			IF fbListClosed.LUIDInList(ipEachPathAhead.StationDestination.LUID) THEN
				// if the successor node is already on the closed list - do nothing, repeate WHILE loop
				CONTINUE;
			END_IF
			
			//Calculate distance to start oh the new found station
			fPathLength := ipActiveStationAStar.PathLength + ipEachPathAhead.Length;
		
			//Check if this station is allready existin in open list - compare if this one is shorter
			IF __QUERYINTERFACE( fbListOpen.FindLUID(ipEachPathAhead.StationDestination.LUID), ipPathFoundInOpenList)  THEN
				IF ipPathFoundInOpenList.PathLength <= fPathLength  THEN
					//object in open list is shorter - do nothing, repeate WHILE loop
					CONTINUE;
				ELSE
					//new object is shorter - remove old object in open lsit
					fbListOpen.RemoveObject(ipPathFoundInOpenList);
				END_IF
			END_IF			
			
			
			//Add this path ahead to open list - set new length
			__QUERYINTERFACE(fbListNotUsedNodes.GetNextObject(), ipEmptyPathObj);
			ipEmptyPathObj.Station := ipEachPathAhead.StationDestination;
			ipEmptyPathObj.RouteUsedToNode.Duplicate(ipActiveStationAStar.RouteUsedToNode);
			ipEmptyPathObj.RouteUsedToNode.AddObject(ipEachPathAhead);
			fbListOpen.AddObject(ipEmptyPathObj);

		END_WHILE
		ipActiveStationAStar.Station.PathsAhead.RestoreIterator();

	END_IF

END_WHILE


//Return station or nothing
IF ipBesStationAStar = 0 THEN
	GetPathToTarget := 0;
ELSE
	//store list in an instance
	fbLastFoundResult.Station := ipBesStationAStar.Station;
	fbLastFoundResult.RouteUsedToNode.Duplicate(ipBesStationAStar.RouteUsedToNode);
	GetPathToTarget := fbLastFoundResult;
END_IF
END_METHOD

METHOD PROTECTED GetPosOnTrack : HRESULT
VAR
	fbPositionXYC : PositionXYC;
END_VAR
//GetArcLengthClosestTo track
THIS^.fPositionOnTrack := THIS^.ipAccocietedTrack.PlanarTrack.GetArcLengthClosestTo(geometry:= THIS^.fbPositionPlanned);

//Get the XYC Pos on track
THIS^.ipAccocietedTrack.PlanarTrack.GetPositionAt(THIS^.PositionOnTrack, fbPositionXYC);

//XYC -> XY
THIS^.fbPositionOnTrackXY.SetValuesXY(fbPositionXYC.x,fbPositionXYC.y);


//Check for NaN
IF NOT(THIS^.fPositionOnTrack = THIS^.fPositionOnTrack) THEN
	GetPosOnTrack := E_FAIL;
	RETURN;
END_IF
END_METHOD

METHOD PROTECTED GetStationAhead : HRESULT
VAR
	ipPath 		: I_XP_Path;
END_VAR
fbStationsAhead.Clear();


fbListPathAhead.ResetIterator();
WHILE fbListPathAhead.HasNextObject() DO
	IF __QUERYINTERFACE(fbListPathAhead.GetNextObject(),ipPath) THEN
		//add StationDestination to list
		fbStationsAhead.AddObject(ipPath.StationDestination);
	END_IF
END_WHILE
END_METHOD

METHOD PROTECTED GetStationBehinde : HRESULT
VAR_INPUT
END_VAR
VAR
	ipThisStation : I_XP_Station;
	ipXpStation : I_XP_Station;
	ipXpStationAhead : I_XP_Station;
END_VAR
ipThisStation := THIS^;
fbStationsBehinde.Clear();

//Check each Station
THIS^.ipXpSystem.StationsUsed.ResetIterator();
WHILE THIS^.ipXpSystem.StationsUsed.HasNextObject() DO
	IF __QUERYINTERFACE(THIS^.ipXpSystem.StationsUsed.GetNextObject(),ipXpStation) THEN
		//check the list of stations ahead if this station one is existing
		ipXpStation.StationsAhead.ResetIterator();
		WHILE ipXpStation.StationsAhead.HasNextObject() DO
			IF __QUERYINTERFACE(ipXpStation.StationsAhead.GetNextObject(),ipXpStationAhead) AND_THEN (ipXpStationAhead = ipThisStation) THEN
				//add station to list
				fbStationsBehinde.AddObject(ipXpStation);
			END_IF
		END_WHILE	
	END_IF
END_WHILE	
THIS^.ipXpSystem.StationsUsed.RestoreIterator();
END_METHOD

METHOD Initialize : HRESULT
VAR
	ipEachStationAhead : I_XP_Station;
	nIdx : UDINT;
END_VAR
VAR_INST
	//This error cannot be reset. Requires a reset cold
	{attribute 'hide'}	
	fbInitError : FB_TcAlarm;
	{attribute 'hide'}	
	fbMissingInterfaceAlarm : FB_TcAlarm;
END_VAR
//Check Error during FB_Init
IF THIS^.bErrorDuringFbInit THEN
	IF NOT fbInitError.bRaised THEN 
		//This error cannot be reset. Requires a reset cold
		fbInitError.CreateEx(stEventEntry:=TC_EVENTS.CHALET_Base_Events.ErrorFBinit, ipSourceInfo := THIS^.fbSourceInfo, bWithConfirmation := FALSE);
		fbInitError.Raise(0);
	END_IF
	Initialize:= E_FAIL;
	THIS^.fbFeedback.HR := Initialize;
	RETURN;
END_IF	

//Interface to System is missing
IF THIS^.ipXpSystem = 0 THEN
	IF NOT fbMissingInterfaceAlarm.bRaised THEN 
		//This error cannot be reset. Requires a reset cold
		fbMissingInterfaceAlarm.CreateEx(stEventEntry:=TC_EVENTS.CHALET_Base_Events.ErrorFBinit, ipSourceInfo := THIS^.fbSourceInfo, bWithConfirmation := FALSE);
		fbMissingInterfaceAlarm.Raise(0);
	END_IF
	Initialize := E_FAIL;
	THIS^.fbFeedback.HR := Initialize;
	RETURN;
END_IF


IF NOT THIS^.bInitDone THEN
	//Busy
	Initialize:= S_PENDING;
	
	//Clean up
	THIS^.DeleteMoversQueue();


	bInitDone := TRUE;
ELSE
	//Done
	Initialize:= S_OK;
END_IF


THIS^.eActiveCommand 				:= CHALET_NC.E_NcAxisCommands.Initialize;
THIS^.fbFeedback.ActiveCommand 		:= TO_STRING(THIS^.eActiveCommand);	
THIS^.fbFeedback.LastCommandAccepted:= TRUE;	
//Set done or keep in busy state	
THIS^.fbFeedback.HR := Initialize;
END_METHOD

METHOD PROTECTED ManageAutomaticallyGeneratedStations : HRESULT
VAR
	ipThisStation : I_XP_Station := THIS^;
	ipTempTrackAhead : I_XP_Track;
	bThisStationIsCreatedAutomatically : BOOL;
	
	bOtherStationsOnThisTrack : BOOL;
	bAnotherTrackAhed : BOOL;
	
	pfbListAllUsedStations : POINTER TO FB_CH_List;
END_VAR
// Check if this station was created by the user, e.g., as a process station, or if it was created automatically at the end of the track to improve track management.
bThisStationIsCreatedAutomatically := (ipThisStation = THIS^.AccocietedTrack.HelperStationAtEndOfTrack);

// Only check automaticali created stations
IF NOT bThisStationIsCreatedAutomatically THEN
	ManageAutomaticallyGeneratedStations := S_OK;
	RETURN;
END_IF



//Set position of this automatic generated station to the end of the accocieted Track
THIS^.PositionXY.x := THIS^.AccocietedTrack.EndPosition.x;
THIS^.PositionXY.y := THIS^.AccocietedTrack.EndPosition.y;



//Check if other Stations are existiong on this track
IF THIS^.AccocietedTrack.StationsOnTrack.Size > 1 THEN
	bOtherStationsOnThisTrack := TRUE;
END_IF

//Another track is before this accocieted track. But the track in front of me is only allowed to have this one track in behind of it.
__QUERYINTERFACE(THIS^.AccocietedTrack.TracksAhead.GetRandomObject(), ipTempTrackAhead);
IF ipTempTrackAhead <> 0 AND_THEN ipTempTrackAhead.TracksBehinde.Size = 1 THEN
	bAnotherTrackAhed := TRUE;
END_IF

//Remove this station from list
/// Todo remove Querypointer - not very OOP
IF (bOtherStationsOnThisTrack OR bAnotherTrackAhed OR NOT XPlanarParameterlist.B_AUTOMATIC_GENARATE_HELPER_STATIONS ) AND __QUERYPOINTER(THIS^.ipXpSystem.StationsUsed, pfbListAllUsedStations) THEN
	//Remove single trackpoint if station is not used
	THIS^.fbOptionalTrackUsedInLiveView.Clear(0);
	pfbListAllUsedStations^.RemoveObject(THIS^);
END_IF
END_METHOD

{attribute 'monitoring':='call'}
PROPERTY MoverAccAtExit : MC_LREAL //[mm/s² on Track] Every mover that leaves or passes the station gets this new acceleration as a target.
GET
MoverAccAtExit := THIS^.fMoverAccAtExit;
END_GET
SET
THIS^.fMoverAccAtExit := MoverAccAtExit;
END_SET
END_PROPERTY

{attribute 'monitoring':='call'}
PROPERTY MoverDecAtExit : MC_LREAL //[mm/s² on Track] Every mover that leaves or passes the station gets this new deceleration as a target.
GET
MoverDecAtExit := THIS^.fMoverDecAtExit;
END_GET
SET
THIS^.fMoverdecAtExit := MoverDecAtExit;
END_SET
END_PROPERTY

{attribute 'monitoring':='call'}
//[mm] Every mover that leaves or passes the station gets this new gap as a target.
PROPERTY MoverGapAtExit : LREAL
GET
MoverGapAtExit := fMoverGapAtExit;
END_GET
SET
IF MoverGapAtExit < XPlanarParameterlist.F_MOVER_MINIMUM_GAP_ON_TRACK THEN
	MoverGapAtExit := XPlanarParameterlist.F_MOVER_MINIMUM_GAP_ON_TRACK;
END_IF

fMoverGapAtExit := MoverGapAtExit;
END_SET
END_PROPERTY

{attribute 'monitoring':='call'}
PROPERTY MoverQueueSize : UINT
GET
MoverQueueSize := THIS^.nMoverQueueSize;
END_GET
SET
THIS^.nMoverQueueSize := MoverQueueSize;
END_SET
END_PROPERTY

{attribute 'monitoring':='call'}
PROPERTY MoversInPlace : BOOL
GET
THIS^.Prepare();//Prepare time-critical information, if not already done


MoversInPlace := bMoversInPlace;
END_GET
END_PROPERTY

{attribute 'monitoring':='call'}
// Return a sorted list of movers in this zone. Index 0 is the mover in Front
PROPERTY MoversInQueue : REFERENCE TO ARRAY [0..(CHALET_BaseComponents.BaseParameterlist.MAX_OBJECTS-1)] OF I_XP_Mover_PLC
GET
MoversInQueue REF= THIS^.fbSortedListMoversInQueue.MoversInZone;
END_GET
END_PROPERTY

{attribute 'monitoring':='call'}
PROPERTY MoverVelocityAtExit : MC_LREAL //[mm/s on Track] Every mover that leaves or passes the station gets this new velocity as a target.
GET
MoverVelocityAtExit := THIS^.fMoverVeloAtExit;
END_GET
SET
THIS^.fMoverVeloAtExit := MoverVelocityAtExit;
END_SET
END_PROPERTY

{attribute 'monitoring':='call'}
//Unique object ID
PROPERTY OID : OTCID
GET
OID := THIS^.fbOptionalTrackUsedInLiveView.MCTOPLC_STD.TrackOID;
END_GET
END_PROPERTY

METHOD PROTECTED OnMoverPasses : BOOL //This methode is called automaticly from the station and detect mover who is passing the station whitout be in queue.
VAR_INPUT
	ipMoverPasses : I_XP_Mover;
END_VAR
VAR
	ipThisStation : I_XP_Station := THIS^;
	
	//this raises an error 33155 "Target position is not reachable. There is no path available to the target position or target position is unreachable in general."
	bPreventMoveCmdToMoversCurrentPos : BOOL;
END_VAR
IF ipMoverPasses = 0 THEN
	RETURN;
END_IF


//Detect mover who is passing the station whitout be in queue. 
//Adjust to new Dynamics
IF NOT THIS^.bSuppressDynamicsChange AND XPlanarParameterlist.B_STATIONS_OVERRIDE_MOVER_DYN_CONSTRAINT THEN
	//Only if not in this queue
	IF ipMoverPasses.ParentStation <> ipThisStation  THEN
		ipMoverPasses.SetDynConstraint_Path(	V:= THIS^.fMoverVeloAtExit, 
												A:= THIS^.fMoverAccAtExit,
												D:= THIS^.fMoverDecAtExit,
												J:= MC_DEFAULT);
	END_IF
END_IF	



//Detect mover who is passing the station whitout be in queue. 
//Adjust to new Gap
IF NOT THIS^.bSuppressDynamicsChange THEN
	bPreventMoveCmdToMoversCurrentPos := (ipMoverPasses.PositionOnTrack = ipMoverPasses.LastCmdTargetPosition) AND (ipMoverPasses.CurrentTrack = ipMoverPasses.LastCmdTargetTrack);
	//Only if not in this queue
	IF ipMoverPasses.ParentStation <> ipThisStation AND NOT bPreventMoveCmdToMoversCurrentPos THEN
		ipMoverPasses.MoveOnTrack(ipTrack	:= ipMoverPasses.LastCmdTargetTrack,
								fPosition	:= ipMoverPasses.LastCmdTargetPosition, 
								fGap		:= THIS^.fMoverGapAtExit);
	END_IF
END_IF
END_METHOD

{attribute 'monitoring':='call'}
//List of paths that lead to stations before this station
PROPERTY PathsAhead : I_CH_List
GET
PathsAhead := THIS^.fbListPathAhead;
END_GET
END_PROPERTY

{attribute 'monitoring':='call'}
//List of paths that lead to stations behind this station
PROPERTY PathsBehinde : I_CH_List
GET
PathsBehinde := THIS^.fbListPathBehind;
END_GET
END_PROPERTY

{attribute 'monitoring':='call'}
//[mm] from the beginning of the assigned track
PROPERTY PositionOnTrack : LREAL
GET
PositionOnTrack := THIS^.fPositionOnTrack;
END_GET
END_PROPERTY

{attribute 'monitoring':='call'}
//Position on the assigned track
PROPERTY PositionOnTrackXY : REFERENCE TO PositionXY
GET
PositionOnTrackXY REF= THIS^.fbPositionOnTrackXY;
END_GET
END_PROPERTY

{attribute 'monitoring':='call'}
//Position on the assigned track
PROPERTY PositionOnTrackXYZABC : REFERENCE TO MoverVector
GET
VAR_INST
	{attribute 'hide'}
	stPosOnTrack : MoverVector;
END_VAR
stPosOnTrack.x := fbPositionOnTrackXY.x;
stPosOnTrack.y := fbPositionOnTrackXY.y;
stPosOnTrack.z := 0;
stPosOnTrack.a := 0;
stPosOnTrack.b := 0;
stPosOnTrack.c := 0;

PositionOnTrackXYZABC REF= stPosOnTrack;
END_GET
END_PROPERTY

{attribute 'monitoring':='call'}
//Planned position, not necessarily on the track. Only changeable when the system is disabled
PROPERTY PositionXY : REFERENCE TO  PositionXY
GET
PositionXY REF= THIS^.fbPositionPlanned;
END_GET
END_PROPERTY

(* 
	Use this Methode to calculate time sensitive date once each cycle. Example: read analog input and convert before do get Signal propertie
*)
METHOD PROTECTED Prepare : HRESULT
VAR_INST
	{attribute 'hide'}	
	nLastUpdatedCycleCount : UDINT;
END_VAR

VAR
	nLoopIndex : UINT;
	fExpectedDistanceToParent : LREAL;
	nCycleTime_ms : UDINT;
	bMoverInQueue : BOOL;
	bTempMoverInPosition : BOOL;
	bTempMoverVeloZero : BOOL;
	bTempMoverInMonitoringTime : BOOL;
	bTempMoverThisStationAsTarget : BOOL;
END_VAR
VAR_INST
	{attribute 'hide'}
	nCycleCountInPos : UDINT;
END_VAR
//Check if this Cycle the dates are allready prepared. This is important for time sensitive informations.
IF nLastUpdatedCycleCount <> TwinCAT_SystemInfoVarList._TaskInfo[THIS^.TaskIndex].CycleCount THEN
	nLastUpdatedCycleCount := TwinCAT_SystemInfoVarList._TaskInfo[THIS^.TaskIndex].CycleCount ;


	(* Check if mover is in place. Time and Position window *)
	//If queuesize is zero, mover is never in place.
	IF nMoverQueueSize = 0 OR THIS^.ipAccocietedTrack = 0 OR NOT ipXpSystem.Enabled THEN
		THIS^.bMoversInPlace := FALSE;
		nCycleCountInPos := 0;
	ELSE
		//Get this task cycle Count and time 
		nCycleTime_ms := TwinCAT_SystemInfoVarList._TaskInfo[THIS^.nTaskIndex].CycleTime(*100ns*) / 10_000 ;
		
		bTempMoverInPosition := TRUE; bTempMoverVeloZero := TRUE; bTempMoverThisStationAsTarget := TRUE;
		fExpectedDistanceToParent := 0;
		FOR nLoopIndex := 0 TO (THIS^.nMoverQueueSize-1) DO
			IF THIS^.fbSortedListMoversInQueue.MoversInZone[nLoopIndex] <> 0 THEN
				//Check position and Gap - 1 mover do not have a gap
				IF nLoopIndex <> 0 THEN
					fExpectedDistanceToParent := fExpectedDistanceToParent + THIS^.fbSortedListMoversInQueue.MoversInZone[nLoopIndex].LastCmdTargetGap;
				END_IF
				bMoverInQueue		:= TRUE;
				bTempMoverInPosition := bTempMoverInPosition AND (ABS(THIS^.fbSortedListMoversInQueue.MoversInZone[nLoopIndex].DistToParentStation - fExpectedDistanceToParent) <= fTargetPosWindow );
				bTempMoverVeloZero := bTempMoverVeloZero AND (THIS^.fbSortedListMoversInQueue.MoversInZone[nLoopIndex].PlanarMover.MCTOPLC.SETONTRACK.SetVelo = 0.0);
				bTempMoverThisStationAsTarget := bTempMoverThisStationAsTarget AND ((THIS^.fbSortedListMoversInQueue.MoversInZone[nLoopIndex].TargetStation = THIS^.TargetGroupe) OR (THIS^.fbSortedListMoversInQueue.MoversInZone[nLoopIndex].TargetStation = THIS^.LUID));
			ELSE
				//Missing mover in queue
				bMoverInQueue := FALSE;
				EXIT;
			END_IF
		END_FOR
			
		//start time if mover position is ok
		IF bTempMoverInPosition  THEN
			nCycleCountInPos := nCycleCountInPos + 1;
		ELSE
			nCycleCountInPos := 0;
		END_IF
		
		bTempMoverInMonitoringTime := (UDINT_TO_TIME(nCycleCountInPos * nCycleTime_ms) >= tTargetPosMonitoringTime);
				
		THIS^.bMoversInPlace := bMoverInQueue AND bTempMoverInPosition AND bTempMoverInMonitoringTime AND bTempMoverThisStationAsTarget;// AND bTempMoverVeloZero;
	END_IF
	
	
END_IF
END_METHOD

{attribute 'monitoring':='call'}
PROPERTY ProcessSimulationActive : BOOL
GET
ProcessSimulationActive := THIS^.fSimulationProcessDuration > 0;
END_GET
END_PROPERTY

//The movers currently in this station must leave the station. 
//The movers actively search for a destination, but only leave if a new destination is available.
METHOD PushMoversOutOfStation : HRESULT
VAR_INPUT
END_VAR
THIS^.nCtsMoversMustLeaveThisStation := THIS^.CtsMoversInQueue;
END_METHOD

{attribute 'monitoring':='call'}
//prevent further movers from entering the station, 
//e.g. to prevent a collision. All movers that are already moving to reach this station will be stopped with a stop 
//and restarted with Ready True.
PROPERTY ReadyToRecvMovers : BOOL
GET
ReadyToRecvMovers := bReadyToRecvMovers;
END_GET
SET
VAR
	ipEachMover : I_XP_Mover;
END_VAR
(* zzz Todo braucht es das?
//Change to Not Ready:
IF (ReadyToRecvMovers = FALSE) AND (bReadyToRecvMovers <> ReadyToRecvMovers) THEN
	//halt all movers on the way
	fbAssignedMovers.ResetIterator();
	WHILE fbAssignedMovers.HasNextObject() DO
		IF ToXpMover(fbAssignedMovers.GetNextObject(),ipEachMover) THEN
			ipEachMover.Halt();	
		END_IF	
	END_WHILE
END_IF

//Change to Ready:
IF (ReadyToRecvMovers = TRUE) AND (bReadyToRecvMovers <> ReadyToRecvMovers) THEN
	//all movers that are on the way have probably been stopped before. when reactivated, the last move command is sent again.
	fbAssignedMovers.ResetIterator();
	WHILE fbAssignedMovers.HasNextObject() DO
		IF ToXpMover(fbAssignedMovers.GetNextObject(),ipEachMover) THEN
			ipEachMover.MoveOnTrack(ipTrack 	:= ipEachMover.LastCmdTargetTrack ,
									fPosition	:= ipEachMover.LastCmdTargetPosition,
									fGap		:= ipEachMover.LastCmdTargetGap);
		END_IF	
	END_WHILE
END_IF
*)
//Store new status
bReadyToRecvMovers := ReadyToRecvMovers;
END_SET
END_PROPERTY

METHOD SendMoversToStation : I_CH_Feedback //All movers in the station are sent to this destination
VAR_INPUT
	sTargetStation: STRING;//unique station name or group of stations
END_VAR
VAR
	nIdx : UDINT;
	ipXpMover : I_XP_Mover;
END_VAR
IF THIS^.fbFeedback.Error THEN
	//Error active/not ready
	THIS^.fbFeedback.LastCommandAccepted	:= FALSE;
	RETURN;
END_IF


//Invalide target
IF sTargetStation = '' THEN
	THIS^.fbFeedback.LastCommandAccepted	:= FALSE;
	RETURN;
END_IF


//Send all Queued movers away by changing the target station destination
THIS^.fbAssignedMovers.ResetIterator();
WHILE THIS^.fbAssignedMovers.HasNextObject() DO
	IF __QUERYINTERFACE(THIS^.fbAssignedMovers.GetNextObject(), ipXpMover) THEN
		
		ipXpMover.TargetStation := sTargetStation;	
		
	END_IF
END_WHILE
THIS^.fbAssignedMovers.RestoreIterator();


//A mover must leave the station immediately when the ‘SendMoversToStation’ method is called. The station is then available again.
//Otherwise, if no destination station is available, the mover waits in the station.
IF XPlanarParameterlist.B_MOVER_MUST_LEAVE_STATION_AT_SET_NEW_TARGED THEN
	//Mover must leave this station
	THIS^.PushMoversOutOfStation();
END_IF



SendMoversToStation := THIS^.fbFeedback;
END_METHOD

METHOD SetTrackObjName : HRESULT
VAR
	ipComObject : ITComObject;
	sName : STRING;
END_VAR
FW_ObjMgr_GetObjectInstance(oid:= THIS^.fbOptionalTrackUsedInLiveView.MCTOPLC_STD.TrackOID, iid:= TC_GLOBAL_IID_LIST.IID_ITComObject, pipUnk:= ADR(ipComObject));
IF ipComObject <> 0 THEN
	sName := THIS^.LUID;
	ipComObject.TcSetObjectName(ADR(sName));
	FW_SafeRelease(ADR(ipComObject));
END_IF
END_METHOD

//If a valid time (>0seconds) is set and the configured destination station exists, then the movers will be sent away automatically after this time from now on.
METHOD SimulationStart : HRESULT
VAR_INPUT
	fProcessDuration 		: LREAL; //[s]
	sTargetStation	: STRING; //Group of the target station to automatic send after the duration
END_VAR
VAR
	ipStation	: I_CH_Object;
	ipXpSystemPlc : I_XP_System_PLC;
	bValideStation : BOOL;
END_VAR
bValideStation := __QUERYINTERFACE(THIS^.ipXpSystem,ipXpSystemPlc) AND ipXpSystemPlc <> 0 AND_THEN ipXpSystemPlc.CheckTargetExists(sTargetStation);

IF (fProcessDuration > 0) AND bValideStation THEN
	//Valide config
	THIS^.fSimulationProcessDuration 	:=	fProcessDuration;
	THIS^.sSimulationTargetStation 		:=	sTargetStation;
	SimulationStart := S_OK;
ELSE
	//Simulation disabled
	THIS^.fSimulationProcessDuration 	:=	0;
	THIS^.sSimulationTargetStation 		:=	'';
	SimulationStart := S_FALSE;
END_IF
END_METHOD

//If a valid time (>0seconds) is set and the configured destination station exists, then the movers will be sent away automatically after this time from now on.
METHOD SimulationStartEx : HRESULT
VAR_INPUT
	fProcessDuration 		: LREAL; //[s]
	ipStation				: I_XP_Station_PLC; //unique station to automatic send after the duration
END_VAR
VAR
	ipXpSystemPlc : I_XP_System_PLC;
	bValideStation : BOOL;
END_VAR
IF ipStation <> 0 THEN
	SimulationStartEx := THIS^.SimulationStart(fProcessDuration := fProcessDuration, sTargetStation := ipStation.LUID);

ELSE
	SimulationStartEx := S_FALSE;
END_IF
END_METHOD

METHOD SimulationStop : HRESULT
//Simulation disabled
THIS^.fSimulationProcessDuration 	:=	0;
THIS^.sSimulationTargetStation 		:=	'';
END_METHOD

{attribute 'monitoring':='call'}
//List of stations before this station
PROPERTY StationsAhead : I_CH_List
GET
StationsAhead := THIS^.fbStationsAhead;
END_GET
END_PROPERTY

{attribute 'monitoring':='call'}
//List of stations behinde this station
PROPERTY StationsBehinde : I_CH_List
GET
StationsBehinde := THIS^.fbStationsBehinde;
END_GET
END_PROPERTY

{attribute 'monitoring':='call'}
//Suppress to change the dynamic(Gap+velocity) of passing movers. This is usefull in startup
PROPERTY SuppressDynamicsChange : BOOL
GET
SuppressDynamicsChange := bSuppressDynamicsChange;
END_GET
SET
bSuppressDynamicsChange := SuppressDynamicsChange;
END_SET
END_PROPERTY

{attribute 'monitoring':='call'}
//Interface to CHALET system to which this object belongs
PROPERTY System : I_XP_System_PLC
GET
//get I_x_System_PLC interface from I_x_System_Registration
__QUERYINTERFACE(THIS^.ipXpSystem, System);
END_GET
END_PROPERTY

{attribute 'monitoring':='call'}
PROPERTY TargetGroupe : STRING
GET
TargetGroupe := THIS^.sTargetGroup;
END_GET
END_PROPERTY

{attribute 'monitoring':='call'}
//A time that is waited as soon as the mover is in the station (including the monitoring window) before “MoversInPlace” is set. e.g. used to stabilize the workpiece
PROPERTY TargetPosMonitoringTime : TIME
GET
TargetPosMonitoringTime := tTargetPosMonitoringTime;
END_GET
SET
tTargetPosMonitoringTime := TargetPosMonitoringTime;
END_SET
END_PROPERTY

{attribute 'monitoring':='call'}
//How many mm before the mover reaches the position is “MoversInPlace” set for the process. 
//This distance can also be set very large (e.g. 100mm) for moving past without stopping.
PROPERTY TargetPosWindow : LREAL
GET
TargetPosWindow := fTargetPosWindow;
END_GET
SET
fTargetPosWindow := TargetPosWindow;
END_SET
END_PROPERTY

METHOD Update : HRESULT
VAR
	nIdx : UDINT;
	bStationIsBlocked : BOOL;
	ipThisStation : I_XP_Station := THIS^;
END_VAR
//Force to do init befor call update
IF NOT bInitDone THEN
	THIS^.Initialize();
	RETURN;
END_IF

THIS^.Prepare();//Prepare time-critical information, if not already done


// ********************** Set feedback depending on active command *******************************
CASE THIS^.eActiveCommand OF

	E_NcAxisCommands.Initialize:
		fbFeedback.Busy 			:= NOT THIS^.bInitDone;
		fbFeedback.Done 			:= THIS^.bInitDone;
		fbFeedback.ErrorId 			:= 0;
		                        	

	ELSE//External command in subclass
		;
END_CASE


// **********************  Stop to execute commands on .done or .error ***************************
IF fbFeedback.Done OR THIS^.fbFeedback.Error THEN
	eActiveCommand 				:= E_NcAxisCommands.None;
END_IF



// **********************  OnMoverPasses ***************************
// Detect mover who is passing the station and call method for easier overwriting
IF fbTrigger.MoverDetected AND (fbTrigger.MoverAtTrigger <> 0) AND_THEN (fbTrigger.MoverAtTrigger.ParentStation <> ipThisStation) THEN
	THIS^.OnMoverPasses(fbTrigger.MoverAtTrigger);
END_IF


// **********************  If enabled start station logic ***************************
IF THIS^.ipXpSystem.Enabled THEN
	
	// Process Simulation. 	
	// All functionality packed into one method for easier overwriting
	THIS^.UpdateSimulation();
	
		
	// Interaction with the movers. Sending on to the next station. 
	// All functionality packed into one method for easier overwriting
	THIS^.UpdateMoverInteraction();
	
	
	//Check for errors
	(*The station is blocked. 
	The first mover in the row is correctly positioned in the station. 
	The queue has a size of >1, but now the n+1 mover does not have this station as its destination. 
	However, it cannot overtake. The station never gives the process a ready signal.*)
	IF THIS^.MoverQueueSize > 1 AND THIS^.MoversInQueue[0] <> 0 AND_THEN (THIS^.MoversInQueue[0].TargetStation = THIS^.TargetGroupe OR THIS^.MoversInQueue[0].TargetStation = THIS^.LUID) THEN
		FOR nIdx := 1 TO (CHALET_BaseComponents.BaseParameterlist.MAX_OBJECTS-1) DO
			//Search for Mover with a direrent target
			IF THIS^.MoversInQueue[nIdx] <> 0 AND_THEN NOT(THIS^.MoversInQueue[nIdx].TargetStation = THIS^.TargetGroupe OR THIS^.MoversInQueue[nIdx].TargetStation = THIS^.LUID) THEN
				//Error
				bStationIsBlocked := TRUE;
				IF NOT fbAlarmStationIsBlocked.bRaised THEN
					//Station is blocked. Mover {0} has {1} as target position but cannot overtake
					fbAlarmStationIsBlocked.CreateEx(TC_Events.CHALET_XPlanar_Events.StationIsBlocked,0,THIS^.fbSourceInfo);
					fbAlarmStationIsBlocked.ipArguments.AddStringByValue(THIS^.MoversInQueue[nIdx].LUID).AddStringByValue(THIS^.MoversInQueue[nIdx].TargetStation);
					fbAlarmStationIsBlocked.Raise(0);
					EXIT;					
				END_IF
			END_IF
		END_FOR
	END_IF
	IF NOT bStationIsBlocked AND fbAlarmStationIsBlocked.bRaised THEN
		fbAlarmStationIsBlocked.Clear(0,0);
	END_IF
	
	
END_IF



// **********************  If disabled clear some bits ***************************
IF NOT THIS^.ipXpSystem.Enabled THEN
	fbAlarmStationIsBlocked.Clear(0,0);
END_IF

Update := S_OK;
END_METHOD

METHOD PROTECTED UpdateMoverInteraction : HRESULT
VAR
	ipFirstMoverInQueue: I_XP_Mover;
	sTargetStation : STRING;
	bMoverValideToSendAway : BOOL;
	bInReachForNewCmd : BOOL;
	bThisStationAsParent : BOOL;
	bFilterDoesNotAllowThisMover : BOOL;
	bThisStationAsTarget : BOOL;
	bMoverIsNotOnAWaitingStation : BOOL;
	bStationInBlockedTryToSolve : BOOL; //Send 1. Mover away ignore that already in correct station
	bMoverMustLeaveTheStation : BOOL; //Set from external
	bSearchNewDestination : BOOL;
	bStationCanBeReachedWhitoutBranch : BOOL;
	bStationIsOverfilled : BOOL;

	ipStationAhead : I_XP_Station;
	ipPathFoundAStarValide : I_PathAStarNode;
	ipPathFoundAStarAnyStation : I_PathAStarNode;
	ipRouteUsed : I_XP_Path;
	
	fbListOf : FB_AStarNode;
	
	
	ipThisStation : I_XP_Station := THIS^;
	ipPath : I_XP_Path;
	ipRoute : I_CH_List;
	ipMover : I_XP_Mover;
	fDistToThisStation : LREAL;
	bValideStationToStartMove : BOOL;
	bValideInterface, bMoverOnSameTrack, bInDecisionDistance : BOOL;
END_VAR
//Get first mover in this station
IF __QUERYINTERFACE(THIS^.MoversInQueue[0],ipFirstMoverInQueue) THEN

	//Get a few helpful variables
	sTargetStation := ipFirstMoverInQueue.TargetStation;
	bThisStationAsTarget := (sTargetStation = THIS^.TargetGroupe) OR (sTargetStation = THIS^.LUID); 
	bThisStationAsParent := ipFirstMoverInQueue.ParentStation.LUID = THIS^.LUID;
	bMoverIsNotOnAWaitingStation := NOT(bThisStationAsParent AND NOT bThisStationAsTarget AND (THIS^.MoverQueueSize > 0));
	bInReachForNewCmd	:= (ipFirstMoverInQueue.DistToParentStation <= THIS^.fDecisionDistance);	
	bStationInBlockedTryToSolve  := THIS^.fbAlarmStationIsBlocked.bRaised;//Send 1. Mover away ignore that already in correct station
	bFilterDoesNotAllowThisMover := (THIS^.Filter <> XPlanarParameterlist.S_ANY_STATION_NAME) AND (THIS^.Filter <> sTargetStation);
	bMoverMustLeaveTheStation := THIS^.nCtsMoversMustLeaveThisStation > 0;
	bStationIsOverfilled  := THIS^.CtsMoversInQueue > THIS^.nMoverQueueSize;
	
	
	//Decide what happens to the mover
	bSearchNewDestination := bInReachForNewCmd AND bThisStationAsParent AND (NOT bThisStationAsTarget OR bMoverMustLeaveTheStation OR bStationInBlockedTryToSolve OR bStationIsOverfilled);
	IF bSearchNewDestination THEN

	
		//1. Prio - Get a direct path to target - Only if specific
		IF sTargetStation <> XPlanarParameterlist.S_ANY_STATION_NAME THEN
			ipPathFoundAStarValide := GetPathToTarget(sTargetStation := sTargetStation);
		END_IF
	
		
		
		//If path to target is not valide, calculate once a path to any station
		IF ipPathFoundAStarValide = 0 THEN
			ipPathFoundAStarAnyStation := THIS^.GetPathToTarget(sTargetStation := XPlanarParameterlist.S_ANY_STATION_NAME);
		END_IF
		
		
		//2. Prio If the next possible station is on this track, without having to pass a switch, then go to this new station
		// The mover should be pushed as far forward as possible to avoid blocking the track
		IF  ipPathFoundAStarValide = 0 AND ipPathFoundAStarAnyStation <> 0  AND (THIS^.PathsAhead.Size = 1) AND THIS^.bNetworkHasTrackBranches THEN
			//
			ipPathFoundAStarAnyStation.RouteUsedToNode.ResetIterator();
			bStationCanBeReachedWhitoutBranch := TRUE;
			WHILE (ipPathFoundAStarAnyStation.RouteUsedToNode.HasNextObject() AND bStationCanBeReachedWhitoutBranch) DO
				IF __QUERYINTERFACE(ipPathFoundAStarAnyStation.RouteUsedToNode.GetNextObject(), ipRouteUsed) THEN
					bStationCanBeReachedWhitoutBranch := (ipRouteUsed.StationDestination.PathsAhead.Size = 1) OR (ipRouteUsed.StationDestination = ipPathFoundAStarAnyStation.Station); //Ignore if destination station have more than 1 paths ahead
				END_IF
			END_WHILE	
			ipPathFoundAStarAnyStation.RouteUsedToNode.RestoreIterator();
			IF bStationCanBeReachedWhitoutBranch THEN
				ipPathFoundAStarValide := ipPathFoundAStarAnyStation;
			END_IF
		END_IF
	
		
		//3. Prio - Send the mover to any station. (most time waitingstation)
		// - closest waitingstation to this station, if not allready on a waiting station
		// - if filter was maybe changed or the mover is not allowed in this station
		IF  ipPathFoundAStarValide = 0 AND ipPathFoundAStarAnyStation <> 0 AND (bMoverIsNotOnAWaitingStation OR bFilterDoesNotAllowThisMover OR bMoverMustLeaveTheStation OR bStationIsOverfilled) THEN
			ipPathFoundAStarValide := ipPathFoundAStarAnyStation;
		END_IF
	END_IF
	
	
	//Write new paths and parent-station to mover
	IF ipPathFoundAStarValide <> 0 THEN 
		//Handover list of paths to mover
		ipFirstMoverInQueue.SetRouteToParent(ipPathFoundAStarValide.RouteUsedToNode);
	
		//Unregister from this station and register with a new parrent station
		THIS^.fbAssignedMovers.RemoveObject(ipFirstMoverInQueue);
		ipPathFoundAStarValide.Station.AddMoverToQueue(ipFirstMoverInQueue);	
		
		//Mover is now leaving the station
		IF THIS^.nCtsMoversMustLeaveThisStation > 0 THEN
			THIS^.nCtsMoversMustLeaveThisStation := THIS^.nCtsMoversMustLeaveThisStation - 1;
		END_IF
		
	END_IF     
END_IF



//---------------------------------------------------------------
//- Update movers not in this queue unsig the route informations
//---------------------------------------------------------------

//The movers have a list of waypoints that they have to travel to on the way to the destination station. 
//It is checked whether this station is one of these waypoints
// - if yes, send the mover to the next waypoint and remove this stop from the list
//Do not wait until mover is at station possition, use fDecisionDistance
ipXpSystem.MoversPresent.ResetIterator();
WHILE ipXpSystem.MoversPresent.HasNextObject() DO
	IF __QUERYINTERFACE(ipXpSystem.MoversPresent.GetNextObject(),ipMover) THEN
		ipRoute := ipMover.RouteRemaining;
		bValideInterface 	:= ipRoute <> 0;
		bMoverOnSameTrack 	:= ipMover.CurrentTrack = ipThisStation.AccocietedTrack;
		fDistToThisStation  := F_GetDistToPosModulo(fTargetPosition := ipThisStation.PositionOnTrack, fActualPosition := (ipMover.PositionOnTrack-1.0), fModulo :=ipThisStation.AccocietedTrack.Length); 
		bInDecisionDistance := (fDistToThisStation <= THIS^.fDecisionDistance);
	ELSE 
		CONTINUE;
	END_IF		
	
	IF bValideInterface AND bMoverOnSameTrack AND bInDecisionDistance THEN
		ipRoute.ResetIterator();
		WHILE ipRoute.HasNextObject() DO
			IF __QUERYINTERFACE(ipRoute.GetNextObject(), ipPath) AND_THEN ipPath.StationStart = ipThisStation THEN
				//Remove this path from route and send to path desination
				ipMover.RouteSegmentDone(ipPath);
				
				//This is normal behavior if not a parent station. 
				//The mover is ~fDecisionDeistance away from the station and is given a new target position to travel further without reducing speed
				IF (fDistToThisStation > 1.0) THEN
					ipMover.MoveOnTrackToStation(ipStation := ipPath.StationDestination,
												fGap:= ipMover.LastCmdTargetGap);
				END_IF	
				 
				 
				//If the mover is very close to the transition, the next settings are already used here
				//This is the case if the mover was in a station for an interaction.
				IF (fDistToThisStation <= 1.0) THEN
					//Set new dynamic. Be careful when reducing the deceleration so that the mover can still stop in real time
					IF XPlanarParameterlist.B_STATIONS_OVERRIDE_MOVER_DYN_CONSTRAINT THEN
						ipMover.SetDynConstraint_Path(	V:= THIS^.fMoverVeloAtExit, 
														A:= THIS^.fMoverAccAtExit,
														D:= THIS^.fMoverDecAtExit,
														J:= MC_DEFAULT);
					END_IF
					ipMover.MoveOnTrackToStation(	ipStation := ipPath.StationDestination,
													fGap := THIS^.fMoverGapAtExit);	
				END_IF	
			END_IF
		END_WHILE
		ipRoute.RestoreIterator();
	END_IF		
END_WHILE
ipXpSystem.MoversPresent.RestoreIterator();
END_METHOD

METHOD PROTECTED UpdateSimulation : HRESULT
VAR_INST
	tonSimulationDelay : TON;
END_VAR
//Automatic send mover to next station in Simulation
//If a valid time (>0seconds) is set and the configured destination station exists, then the movers will be sent away automatically after this time from now on.
tonSimulationDelay.IN 	:= THIS^.ipXpSystem.Enabled AND THIS^.MoversInPlace AND THIS^.ProcessSimulationActive;
tonSimulationDelay.PT	:= LREAL_TO_TIME(THIS^.fSimulationProcessDuration*1000.0);
tonSimulationDelay();
IF tonSimulationDelay.Q THEN
	THIS^.SendMoversToStation(sTargetStation := THIS^.sSimulationTargetStation);
END_IF
END_METHOD

END_FUNCTION_BLOCK

// ---- COMPONENTs/Environment/FB_XP_Environment.TcPOU
{attribute 'no_explicit_call' := 'Do not call the body - Stick to OOP'}
(* XPlanar Environment - 1 per associated XPlanar 
	The Planar environment is a software object that represents the two-dimensional XPlanar stator surface. Together with Planar movers in a group, 
	it prevents collisions of the movers with the edge of the surface. *)
FUNCTION_BLOCK FB_XP_Environment EXTENDS FB_CH_Object IMPLEMENTS I_XP_Environment
VAR
	//Link to Planar-Environment object
	fbEnvironment : MC_PlanarEnvironment;
	fbUtilityEnvirement : FB_TcIoXPlanarEnvironment;
	
	{attribute 'hide'}  
	bInitDone :BOOL := FALSE;
	{attribute 'hide'}
	ipXpSystem : I_XP_System_Registration;
	{attribute 'hide'}               	
	fbFeedback 			: FB_XP_Feedback(ipSourceInfo := fbSourceInfo);	
	{attribute 'hide'}                   	
	eActiveCommand 		: CHALET_Nc.E_NcAxisCommands := CHALET_Nc.E_NcAxisCommands.None;
	{attribute 'hide'}
	bCollisionCheckEnabled : BOOL := TRUE;
	{attribute 'hide'}
	fMoverOffsetWarning : LREAL := 2.0; //[mm]
	{attribute 'hide'}
	fMoverOffsetError: LREAL := 0.0;//[mm]
	{attribute 'hide'}
	eMoverDetectionStatus : MoverDetectionStatus;
	{attribute 'hide'}
	eMoverDetectionStatusLastCycle : MoverDetectionStatus;
END_VAR


// Planar-Feedback objects
VAR
	{attribute 'hide'} 
	fbFeedbackAddToGrp : MC_PlanarFeedback;
	{attribute 'hide'} 
	fbFeedbackRmvFromGrp : MC_PlanarFeedback;
	{attribute 'hide'} 
	fbFeedbackConfigure : MC_PlanarFeedback;
	{attribute 'hide'} 
	fbFeedbackClear : MC_PlanarFeedback;
END_VAR

METHOD AddToGroup : HRESULT
VAR_INPUT
	iGroup : I_XP_Group;
END_VAR
IF NOT THIS^.fbFeedback.Busy THEN
	THIS^.eActiveCommand 				:= CHALET_NC.E_NcAxisCommands.AddToGroupe;
	THIS^.fbFeedback.ActiveCommand 		:= TO_STRING(THIS^.eActiveCommand);	
	THIS^.fbFeedback.LastCommandAccepted:= TRUE;		
	THIS^.fbFeedback.Busy 				:= TRUE;
	
	iGroup.AddEnvironment(THIS^.fbEnvironment, THIS^.fbFeedbackAddToGrp);
	AddToGroup := S_OK;
ELSE
	AddToGroup := S_FALSE;
	THIS^.fbFeedback.LastCommandAccepted:= FALSE;	
END_IF
END_METHOD

(* Clears the Planar Environment (stators and boundary). *)
METHOD Clear : HRESULT
THIS^.eActiveCommand 				:= CHALET_NC.E_NcAxisCommands.Clear;
THIS^.fbFeedback.ActiveCommand 		:= TO_STRING(THIS^.eActiveCommand);	
THIS^.fbFeedback.LastCommandAccepted:= TRUE;		
THIS^.fbFeedback.Busy 				:= TRUE;

THIS^.fbEnvironment.Clear(commandFeedback:=THIS^.fbFeedbackClear);
Clear := S_OK;
END_METHOD

{attribute 'monitoring':='call'}
(* If Enable, the movers are checked for collisions with each other.
Warning and error can have their own size offsets.
The error leads to a stop with higher dynamics.
In simulation, an error does not lead to a stop *)
PROPERTY CollisionCheck : BOOL
GET
CollisionCheck := THIS^.bCollisionCheckEnabled;
END_GET
SET
THIS^.bCollisionCheckEnabled := CollisionCheck;
END_SET
END_PROPERTY

//Return an interface to the mover if a collision is active else return 0. The check stops after the first collision found
METHOD PROTECTED CollisionDetectionAlgorithm : I_XP_Mover
VAR_INPUT
	ipListOfMovers : I_CH_LIST;
	fOffsetMoverSize : LREAL := 1.0; //Offset on the mover dimension from the MC3 mover object [mm];
END_VAR
VAR
	aPointsMover1 : ARRAY[0..3] OF  Tc3_Physics.PositionXY;
	aPointsEachMover : ARRAY[0..3] OF  Tc3_Physics.PositionXY;
	aPointsDelta : ARRAY[0..3] OF  Tc3_Physics.PositionXY;
	
	fMoverWidth, fMoverHight : LREAL;
	fMoverXPos, fMoverYPos, fMoverCPos : LREAL;
	
	ipMover1, ipEachMover : I_XP_Mover;
	fbListOfMoverToCheck : FB_CH_List;
	
	fAngle : LREAL;
	a, b, c: LREAL;
	Pa, Pb, Pc : REFERENCE TO Tc3_Physics.PositionXY;
	fcos : LREAL;
	
	nIdx, nIdxMover1, nIdxPlus1 : UINT;
	ipMover2CollisionFound : I_XP_Mover;
END_VAR
//Get all mover in a list
fbListOfMoverToCheck.Duplicate(ipListOfMovers);



//Check list for invalide Act Pos - ex.: if mover is not found 
fbListOfMoverToCheck.ResetIterator();
WHILE fbListOfMoverToCheck.HasNextObject() DO
	__QUERYINTERFACE(fbListOfMoverToCheck.GetNextObject(),ipMover1);
	
	IF ipMover1.MoverIsNotPresent THEN 		
		//remove from list
		fbListOfMoverToCheck.RemoveObject(ipMover1);
		
	END_IF
END_WHILE



fbListOfMoverToCheck.ResetIterator();
WHILE fbListOfMoverToCheck.HasNextObject() DO
	//get first mover in list,
	__QUERYINTERFACE(fbListOfMoverToCheck.GetNextObject(),ipMover1);
	
	fMoverXPos := ipMover1.PositionAct.x;
	fMoverYPos := ipMover1.PositionAct.y;
	fMoverCPos := ipMover1.PositionAct.c;
		
	//Get corner points of the rectangle 
	fMoverWidth := ipMover1.MoverWidth - fOffsetMoverSize;
	fMoverHight := ipMover1.MoverHeight - fOffsetMoverSize;
	aPointsMover1[0].SetValuesXY(x:= -fMoverWidth/2, y:= -fMoverHight/2);//Bottom Left
	aPointsMover1[1].SetValuesXY(x:= -fMoverWidth/2, y:=  fMoverHight/2);//Top Left
	aPointsMover1[2].SetValuesXY(x:=  fMoverWidth/2, y:=  fMoverHight/2);//Top Ritgh
	aPointsMover1[3].SetValuesXY(x:=  fMoverWidth/2, y:= -fMoverHight/2);//Bottom Rigth
	
	//Rotation of the mover
	F_RotatePositionXY(aPointsMover1[0], fMoverCPos);
	F_RotatePositionXY(aPointsMover1[1], fMoverCPos);
	F_RotatePositionXY(aPointsMover1[2], fMoverCPos);
	F_RotatePositionXY(aPointsMover1[3], fMoverCPos);
	
	//shift to mover coordinates
	aPointsMover1[0].ShiftByXY(dx:= fMoverXPos, dy:= fMoverYPos);
	aPointsMover1[1].ShiftByXY(dx:= fMoverXPos, dy:= fMoverYPos);
	aPointsMover1[2].ShiftByXY(dx:= fMoverXPos, dy:= fMoverYPos);
	aPointsMover1[3].ShiftByXY(dx:= fMoverXPos, dy:= fMoverYPos);
	
	
	//do an check for all mover
	fbListOfMoverToCheck.ResetIterator();
	WHILE fbListOfMoverToCheck.HasNextObject() DO
		__QUERYINTERFACE(fbListOfMoverToCheck.GetNextObject(),ipEachMover);
		
		//Skip if same
		IF ipEachMover = ipMover1 THEN
			CONTINUE;
		END_IF
		
		//Skip if far away
		IF (MAX(ipEachMover.MoverHeight, ipEachMover.MoverWidth) + MAX(ipMover1.MoverHeight, ipMover1.MoverWidth) + fOffsetMoverSize) < F_DistXYVectors(ipEachMover.PositionAct, ipMover1.PositionAct) THEN
			CONTINUE;
		END_IF
		
		
		fMoverXPos := ipEachMover.PositionAct.x;
		fMoverYPos := ipEachMover.PositionAct.y;
		fMovercPos := ipEachMover.PositionAct.c;
		
		//Get corner points of the rectangle 
		fMoverWidth := ipEachMover.MoverWidth - fOffsetMoverSize;
		fMoverHight := ipEachMover.MoverHeight - fOffsetMoverSize;
		aPointsEachMover[0].SetValuesXY(x:= -fMoverWidth/2, y:= -fMoverHight/2);//Bottom Left
		aPointsEachMover[1].SetValuesXY(x:= -fMoverWidth/2, y:=  fMoverHight/2);//Top Left
		aPointsEachMover[2].SetValuesXY(x:=  fMoverWidth/2, y:=  fMoverHight/2);//Top Ritgh
		aPointsEachMover[3].SetValuesXY(x:=  fMoverWidth/2, y:= -fMoverHight/2);//Bottom Rigth

		//Rotation of the mover
		F_RotatePositionXY(aPointsEachMover[0], fMoverCPos);
		F_RotatePositionXY(aPointsEachMover[1], fMoverCPos);
		F_RotatePositionXY(aPointsEachMover[2], fMoverCPos);
		F_RotatePositionXY(aPointsEachMover[3], fMoverCPos);
		
		//shift to mover coordinates
		aPointsEachMover[0].ShiftByXY(dx:= fMoverXPos, dy:= fMoverYPos);
		aPointsEachMover[1].ShiftByXY(dx:= fMoverXPos, dy:= fMoverYPos);
		aPointsEachMover[2].ShiftByXY(dx:= fMoverXPos, dy:= fMoverYPos);
		aPointsEachMover[3].ShiftByXY(dx:= fMoverXPos, dy:= fMoverYPos);		
		
		//check each corener if inside each mover
		FOR nIdxMover1 := 0 TO 3 DO
			
			(* A triangle is created between a corner point of Mover1 (point a) and two corner points of Mover2 (points B and C). 
			All corner points of Mover2 are now tested one after the other. If the sum of all angles "a" is 360 degrees, 
			then point A is inside mover 2 and there is a collision *)
			fAngle := 0;
			FOR nIdx := 0 TO 3 DO
				nIdxPlus1 := ((nIdx+1)MOD 4);
			
				Pa REF= aPointsMover1[nIdxMover1];
				Pb REF= aPointsEachMover[nIdx];
				Pc REF= aPointsEachMover[nIdxPlus1];					
				

				a := SQRT(EXPT((Pb.x - Pc.x),2)+EXPT((Pb.y - Pc.y),2));
				b := SQRT(EXPT((Pa.x - Pc.x),2)+EXPT((Pa.y - Pc.y),2));
				c := SQRT(EXPT((Pa.x - Pb.x),2)+EXPT((Pa.y - Pb.y),2));
				
				
				IF b=0 OR c=0 THEN
					//Error - Return the found mover
					CollisionDetectionAlgorithm := ipMover1;
					//with which mover is the collision
					ipMover2CollisionFound := ipEachMover;
					RETURN;
				ELSE
					(*  a/sin(α) = b/sin(β) = c/sin(γ) *)
					fcos := (EXPT(b,2) + EXPT(c,2) - EXPT(a,2))/(2*b*c);
					fcos := LIMIT(-1.0, fcos, 1.0);
					fAngle :=  fAngle + ACOS(fcos);
				END_IF
			END_FOR
			
			//if the point is inside the mover, the sum of all angles is exactly 360°-> 2pi
			IF ABS(fAngle - 2*Tc2_System.PI)<0.01 THEN
				//Error - Return the found mover
				CollisionDetectionAlgorithm := ipMover1;
				//with which mover is the collision
				ipMover2CollisionFound := ipEachMover;
				RETURN;
			END_IF
			
		END_FOR

	END_WHILE
	fbListOfMoverToCheck.RestoreIterator();
	
	
	
END_WHILE
END_METHOD

METHOD Configure : HRESULT
THIS^.eActiveCommand 				:= CHALET_NC.E_NcAxisCommands.Configure;
THIS^.fbFeedback.ActiveCommand 		:= TO_STRING(THIS^.eActiveCommand);	
THIS^.fbFeedback.LastCommandAccepted:= TRUE;		
THIS^.fbFeedback.Busy 				:= TRUE;

THIS^.fbEnvironment.CreateBoundary(commandFeedback:=THIS^.fbFeedbackConfigure);
Configure := S_OK;
END_METHOD

METHOD FB_init : BOOL
VAR_INPUT
	bInitRetains : BOOL; // if TRUE, the retain variables are initialized (warm start / cold start)
	bInCopyCode : BOOL;  // if TRUE, the instance afterwards gets moved into the copy code (online change)
	
	ipSystem : I_CH_Object;
END_VAR
//Do the following code once during start up and not during onlinechange
IF NOT bInCopyCode THEN 
	
	(* Register to the Xplanar System
	   1. Test if the interface exists
	   2. Test if the object implements a "System for Mover" interface 
	*)
	IF ipSystem <> 0 AND_THEN __QUERYINTERFACE(ipSystem,THIS^.ipXpSystem) THEN
		THIS^.ipXpSystem.LinkEnvironment(THIS^);
	END_IF
	
	
	THIS^.fbFeedback.ActiveCommand 		:= TO_STRING(THIS^.eActiveCommand);	
	
END_IF
END_METHOD

{attribute 'monitoring':='call'}
PROPERTY Feedback : I_XP_Feedback
GET
Feedback := THIS^.fbFeedback;
END_GET
END_PROPERTY

METHOD Initialize : HRESULT
VAR
	stVarInfo : __SYSTEM.VAR_INFO;
END_VAR
VAR_INST
	//This error cannot be reset. Requires a reset cold
	{attribute 'hide'}	
	fbInitError : FB_TcAlarm;
END_VAR
// Check if link to envirement is mapped
IF NOT THIS^.Mapped THEN
	IF NOT fbInitError.bRaised THEN 
		//This error cannot be reset. Requires a reset cold
		fbInitError.CreateEx(stEventEntry:=TC_EVENTS.CHALET_Base_Events.VariableLinkMissing, ipSourceInfo := THIS^.fbSourceInfo, bWithConfirmation := FALSE);
		stVarInfo := __VARINFO(fbEnvironment);
		fbInitError.ipArguments.AddString(stVarInfo.Symbol);
		fbInitError.Raise(0);
	END_IF
	Initialize := E_FAIL;
	RETURN;
END_IF



IF NOT bInitDone THEN
	//Busy
	Initialize := S_PENDING;
	
	IF fbUtilityEnvirement.Init(bExecute := TRUE) THEN
		fbUtilityEnvirement.Init(bExecute := FALSE);
		bInitDone := TRUE;
	END_IF
	
	
ELSE	
	//Done
	Initialize := S_OK;
END_IF


THIS^.eActiveCommand 				:= CHALET_NC.E_NcAxisCommands.Initialize;
THIS^.fbFeedback.ActiveCommand 		:= TO_STRING(THIS^.eActiveCommand);	
THIS^.fbFeedback.LastCommandAccepted:= TRUE;	
//Set done or keep in busy state	
THIS^.fbFeedback.HR := Initialize;
END_METHOD

{attribute 'monitoring':='call'}
PROPERTY Mapped : BOOL //Project is mapped to MC (McToPlc and PlcToMc)
GET
VAR
	bMcToPlcNotMapped 	: BOOL;
END_VAR
bMcToPlcNotMapped := F_GetMappingStatus(ADR(THIS^.fbEnvironment.MCTOPLC_STD), SIZEOF(THIS^.fbEnvironment.MCTOPLC_STD)) <> EPlcMappingStatus.MS_Mapped;

Mapped := NOT bMcToPlcNotMapped;
END_GET
END_PROPERTY

{attribute 'monitoring':='call'}
//Offset on the mover dimension from the MC3 mover object [mm] ;
// >0 menas the warning is earlier
PROPERTY MoverCollisionOffsetError : LREAL
GET
MoverCollisionOffsetError := fMoverOffsetError;
END_GET
SET
fMoverOffsetError := MoverCollisionOffsetError;
END_SET
END_PROPERTY

{attribute 'monitoring':='call'}
//Offset on the mover dimension from the MC3 mover object [mm] ;
// >0 menas the warning is earlier
PROPERTY MoverCollisionOffsetWarning : LREAL
GET
MoverCollisionOffsetWarning :=  fMoverOffsetWarning;
END_GET
SET
fMoverOffsetWarning := MoverCollisionOffsetWarning;
END_SET
END_PROPERTY

{attribute 'monitoring':='call'}
//Unique object ID
PROPERTY OID : OTCID
GET
OID := THIS^.fbEnvironment.MCTOPLC_STD.EnvironmentOID;
END_GET
END_PROPERTY

{attribute 'monitoring':='call'}
PROPERTY PlanarEnvironment : REFERENCE TO MC_PlanarEnvironment
GET
PlanarEnvironment ref= THIS^.fbEnvironment;
END_GET
END_PROPERTY

(* Time-critical information is processed here, which can then be polled via the property every cycle. 
The update method is usually at the end of the program and then it is already 'outdated'. *)
METHOD PRIVATE Prepare : HRESULT
VAR CONSTANT
	N_IDX_OFFSET_MoverDetectionStatus 	: UDINT := 16#03171005; // Parameter(online) in Planar  Processing Unit object 
END_VAR
VAR
	nParaSize : UDINT;
	pParaData : PVOID;
	hr : HRESULT;
	ipComObject : ITComObject;
END_VAR
VAR_INST
	{attribute 'hide'}
	nLastUpdatedCycleCount : UDINT;
END_VAR
//Check if this Cycle the dates are allready prepared
IF nLastUpdatedCycleCount <> TwinCAT_SystemInfoVarList._TaskInfo[THIS^.nTaskIndex].CycleCount THEN
	nLastUpdatedCycleCount := TwinCAT_SystemInfoVarList._TaskInfo[THIS^.nTaskIndex].CycleCount;

	
	//************** Read MoverDetectionStatus **************
	//Get interface to ComObject
	FW_ObjMgr_GetObjectInstance(oid:= THIS^.ProcessingUnitOID, iid:= TC_GLOBAL_IID_LIST.IID_ITComObject, pipUnk:= ADR(ipComObject));
	
	//Get ADR and SIZE
	nParaSize := SIZEOF(eMoverDetectionStatus);	pParaData := ADR(eMoverDetectionStatus);
	
	IF ipComObject <> 0 THEN
		hr := ipComObject.TcGetObjPara(pid:=N_IDX_OFFSET_MoverDetectionStatus , nData:= nParaSize, pData:= pParaData, pgp:=0 );	
		FW_SafeRelease(ADR(ipComObject));
	END_IF
	
	//force to have the in progress active FOR 1 cycle longer
	IF eMoverDetectionStatus = MoverDetectionStatus.DetectionSuccessful AND eMoverDetectionStatusLastCycle = MoverDetectionStatus.DetectionInProcess THEN
		//Store info from last cycle
		eMoverDetectionStatusLastCycle := eMoverDetectionStatus;
		eMoverDetectionStatus := MoverDetectionStatus.DetectionInProcess;
	ELSE	
		//Store info from last cycle
		eMoverDetectionStatusLastCycle := eMoverDetectionStatus;
	END_IF
	


		
END_IF
END_METHOD

{attribute 'monitoring':='call'}
//Enumeration MoverDetectionStatus
PROPERTY ProcessingUnitMoverDetectionStatus : MoverDetectionStatus
GET
THIS^.Prepare();//Prepare time-critical information, if not already done


ProcessingUnitMoverDetectionStatus := THIS^.eMoverDetectionStatus;
END_GET
END_PROPERTY

{attribute 'monitoring':='call'}
//Object ID of the IoXPlanar processing unit
PROPERTY ProcessingUnitOID : OTCID
GET
VAR
	nProcessingUnitOid : OTCID;
END_VAR
VAR CONSTANT
	N_IDX_OFFSET_PU_Oid 	: UDINT := 16#050300C0; // Parameter(online) in Planar Environment object 
END_VAR

VAR
	nParaSize : UDINT;
	pParaData : PVOID;
	hr : HRESULT;
	ipComObject : ITComObject;
	nOid : OTCID;
END_VAR
//Get TcCom Object ID
nOid := THIS^.OID;

//Get interface to ComObject
FW_ObjMgr_GetObjectInstance(oid:= nOid, iid:= TC_GLOBAL_IID_LIST.IID_ITComObject, pipUnk:= ADR(ipComObject));

//Get ADR and SIZE
nParaSize := SIZEOF(nProcessingUnitOid);	pParaData := ADR(nProcessingUnitOid);

IF ipComObject <> 0 THEN
	hr := ipComObject.TcGetObjPara(pid:=N_IDX_OFFSET_PU_Oid , nData:= nParaSize, pData:= pParaData, pgp:=0 );	
	FW_SafeRelease(ADR(ipComObject));
END_IF

ProcessingUnitOID := nProcessingUnitOid;
END_GET
END_PROPERTY

METHOD RemoveFromGroup : HRESULT
IF NOT THIS^.fbFeedback.Busy THEN
	THIS^.eActiveCommand 				:= CHALET_NC.E_NcAxisCommands.RemoveFromGroupe;
	THIS^.fbFeedback.ActiveCommand 		:= TO_STRING(THIS^.eActiveCommand);	
	THIS^.fbFeedback.LastCommandAccepted:= TRUE;		
	THIS^.fbFeedback.Busy 				:= TRUE;
	
	THIS^.fbEnvironment.RemoveFromGroup(THIS^.fbFeedbackRmvFromGrp);
	RemoveFromGroup := S_OK;
ELSE
	RemoveFromGroup := S_FALSE;
	THIS^.fbFeedback.LastCommandAccepted:= FALSE;	
END_IF
END_METHOD

{attribute 'monitoring':='call'}
//Interface to CHALET system to which this object belongs
PROPERTY System : I_XP_System_PLC
GET
//get I_x_System_PLC interface from I_x_System_Registration
__QUERYINTERFACE(THIS^.ipXpSystem, System);
END_GET
END_PROPERTY

METHOD PUBLIC Update : HRESULT



// ********************** Set feedback depending on active command *******************************
CASE THIS^.eActiveCommand OF
	E_NcAxisCommands.None: 
		//Display if a Mover Error is active during no command is active
		IF THIS^.fbEnvironment.Error AND NOT fbFeedback.Error THEN 
			fbFeedback.ErrorId 			:= THIS^.fbEnvironment.ErrorID;
			fbFeedback.ActiveCommand 	:= TO_STRING(E_NcAxisCommands.None);	
			fbFeedback.ClearObjectInfo();
		END_IF

	E_NcAxisCommands.Initialize:
		fbFeedback.Busy 			:= NOT THIS^.bInitDone;
		fbFeedback.Done 			:= THIS^.bInitDone;
		fbFeedback.ErrorId 			:= 0;
		fbFeedback.ClearObjectInfo();
		                                                       			                        	
	E_NcAxisCommands.Clear:     	
		fbFeedback.Busy 			:= fbFeedbackClear.Busy;
		fbFeedback.Done 			:= fbFeedbackClear.Done;
		fbFeedback.ErrorId 			:= fbFeedbackClear.ErrorID;
        fbFeedback.ObjectInfo		:= fbFeedbackClear.objectInfo;
           			                        	
	E_NcAxisCommands.Configure:     	
		fbFeedback.Busy 			:= fbFeedbackConfigure.Busy;
		fbFeedback.Done 			:= fbFeedbackConfigure.Done;
		fbFeedback.ErrorId 			:= fbFeedbackConfigure.ErrorID;
        fbFeedback.ObjectInfo		:= fbFeedbackConfigure.objectInfo;
                                      			                        	
	E_NcAxisCommands.AddToGroupe:     	
		fbFeedback.Busy 			:= fbFeedbackAddToGrp.Busy;
		fbFeedback.Done 			:= fbFeedbackAddToGrp.Done;
		fbFeedback.ErrorId 			:= fbFeedbackAddToGrp.ErrorID;
        fbFeedback.ObjectInfo		:= fbFeedbackAddToGrp.objectInfo;
                                      			                        	
	E_NcAxisCommands.RemoveFromGroupe:     	
		fbFeedback.Busy 			:= fbFeedbackRmvFromGrp.Busy;
		fbFeedback.Done 			:= fbFeedbackRmvFromGrp.Done;
		fbFeedback.ErrorId 			:= fbFeedbackRmvFromGrp.ErrorID;
        fbFeedback.ObjectInfo		:= fbFeedbackRmvFromGrp.objectInfo;
                                		
	ELSE//External command in subclass
		;
END_CASE


// **********************  Stop to execute commands on .done or .error ***************************
IF fbFeedback.Done OR THIS^.fbFeedback.Error THEN
	eActiveCommand 				:= E_NcAxisCommands.None;
END_IF





//Update Collision subroutin
THIS^.UpdateCollisionDetection();


//Update xplanar object
THIS^.fbEnvironment.Update();

//Update feedback object
fbFeedbackConfigure.Update(); 
fbFeedbackClear.Update(); 
fbFeedbackAddToGrp.Update(); 
fbFeedbackRmvFromGrp.Update();
END_METHOD

METHOD PROTECTED UpdateCollisionDetection : HRESULT
VAR
	bDisableDuringMoverDetection : BOOL;
	ipMoverCollision : I_XP_Mover;
	ipSystemPlc : I_XP_System_PLC;
	nX, nY : DINT;
END_VAR
VAR_INST
	{attribute 'hide'}	
	ipMoverCollisionOldWarning : I_XP_Mover;
	{attribute 'hide'}	
	fbAlarmCollisionMoverWarning : FB_TcAlarm;	
	{attribute 'hide'}	
	ipMoverCollisionOldAlarm : I_XP_Mover;
	{attribute 'hide'}	
	fbAlarmCollisionMoverAlarm : FB_TcAlarm;
END_VAR
bDisableDuringMoverDetection := THIS^.ProcessingUnitMoverDetectionStatus = MoverDetectionStatus.DetectionInProcess;


//Check whether a mover has a collision with another mover and generate a warning.
//Only 1 mover is found and displayed
//WARNING - each mover default is 2mm larger
IF THIS^.bCollisionCheckEnabled AND NOT bDisableDuringMoverDetection THEN
	//get mover or 0 for no collision
	ipMoverCollision := CollisionDetectionAlgorithm(fOffsetMoverSize := THIS^.fMoverOffsetWarning, ipListOfMovers := THIS^.ipXpSystem.MoversPresent);
	
	IF ipMoverCollision <> 0 AND_THEN ipMoverCollision <> ipMoverCollisionOldWarning AND_THEN NOT ipMoverCollision.MoverIsNotPresent THEN
		fbAlarmCollisionMoverWarning.CreateEx(tc_Events.CHALET_XPlanar_Events.MoverCollisionWarning, 0, THIS^.fbSourceInfo);
		//Mover "{0}" has a collision with another mover at position X:{1} Y:{2}
		nX := LREAL_TO_DINT(ipMoverCollision.PlanarMover.MCTOPLC.ACT.ActPos.x);
		nY := LREAL_TO_DINT(ipMoverCollision.PlanarMover.MCTOPLC.ACT.ActPos.y);
		fbAlarmCollisionMoverWarning.ipArguments.Clear().AddStringByValue(ipMoverCollision.LUID).AddDInt(nX).AddDint(nY);
		fbAlarmCollisionMoverWarning.Raise(0);
	ELSIF ipMoverCollision = 0 THEN
		//No collision found
		fbAlarmCollisionMoverWarning.Clear(0,0);
	END_IF
	ipMoverCollisionOldWarning := ipMoverCollision;
ELSE
	fbAlarmCollisionMoverWarning.Clear(0,0);
	ipMoverCollisionOldWarning := 0;
END_IF

//Check whether a mover has a collision with another mover and generate a warning.
//Only 1 mover is found and displayed
//ERROR - each mover is default -1mm smaller
IF THIS^.bCollisionCheckEnabled AND NOT bDisableDuringMoverDetection  THEN
	//get mover or 0 for no collision
	ipMoverCollision := CollisionDetectionAlgorithm(fOffsetMoverSize := THIS^.fMoverOffsetError, ipListOfMovers := THIS^.ipXpSystem.MoversPresent);
	
	IF ipMoverCollision <> 0 AND ipMoverCollision <> ipMoverCollisionOldAlarm THEN
		fbAlarmCollisionMoverAlarm.CreateEx(tc_Events.CHALET_XPlanar_Events.MoverCollisionStop, 0, THIS^.fbSourceInfo);
		//Mover "{0}" has a collision with another mover at position X:{1} Y:{2}
		fbAlarmCollisionMoverAlarm.ipArguments.AddStringByValue(ipMoverCollision.LUID).AddUDInt(LREAL_TO_UDINT(ipMoverCollision.PlanarMover.MCTOPLC.ACT.ActPos.x)).AddUDInt(LREAL_TO_UDINT(ipMoverCollision.PlanarMover.MCTOPLC.ACT.ActPos.y));
		fbAlarmCollisionMoverAlarm.Raise(0);

		//Stop if this is a real system, keep running in simulation
		
		IF THIS^.UtilityEnvirement.TcIoXpu(1).GetOperationMode() = XplanarOperationMode.Normal THEN
			IF __QUERYINTERFACE(THIS^.ipXpSystem, ipSystemPlc) THEN
				//Disable System
				ipSystemPlc.FastStop();
			END_IF
		END_IF
	ELSIF ipMoverCollision = 0 THEN
		//No collision found
		fbAlarmCollisionMoverAlarm.Clear(0,0);
	END_IF
		
	ipMoverCollisionOldAlarm := ipMoverCollision;
ELSE
	fbAlarmCollisionMoverAlarm.Clear(0,0);
	ipMoverCollisionOldAlarm := 0;
END_IF
END_METHOD

{attribute 'monitoring':='call'}
PROPERTY UtilityEnvirement : Tc3_XPlanarUtility.I_Environment
GET
UtilityEnvirement := fbUtilityEnvirement;
END_GET
END_PROPERTY

END_FUNCTION_BLOCK

// ---- FUNCTIONs/F_RotatePositionXY.TcPOU
FUNCTION F_RotatePositionXY : HRESULT
VAR_INPUT
	fbPosition : REFERENCE TO Tc3_Physics.PositionXY;
	fRotate : LREAL; //[°]
END_VAR
VAR
	fRadius : LREAL;
	fPhi : LREAL;
	fNewPhi : LREAL;
END_VAR

IF NOT __ISVALIDREF(fbPosition) THEN
	F_RotatePositionXY := E_FAIL;
	RETURN;
END_IF

fRadius := fbPosition.GetRadius();
fPhi := fbPosition.GetPhi();

fNewPhi := MODABS((fPhi + fRotate), 360.0);

fbPosition.SetValuesRP(radius := fRadius, phi := fNewPhi);

END_FUNCTION

// ---- COMPONENTs/Group/FB_XP_Group.TcPOU
{attribute 'no_explicit_call' := 'Do not call the body - Stick to OOP'}
(* XPlanar Collision Avoidance Groupe - 1 per associated XPlanar 
	The Planar group is a software object that prevents collisions between Planar movers as well as collisions of Planar movers with the boundary of 
	the stator area on the two-dimensional XPlanar stator area. To do this, the 2D areas of all objects in the group are blocked. When a motion command 
	is transferred to a mover, the required area is requested from the Planar group and the motion command is rejected if this area would collide 
	with already reserved areas. If the motion command can be executed, the area is added to the set of reserved area and blocked accordingly. *)
FUNCTION_BLOCK FB_XP_Group EXTENDS FB_CH_Object IMPLEMENTS I_XP_Group
VAR
	//Link to Planar-Group object
	fbGroup : MC_PlanarGroup;
		
	{attribute 'hide'}  
	bInitDone :BOOL := FALSE;
	{attribute 'hide'}
	ipXpSystem : I_XP_System_Registration;
	{attribute 'hide'}               	
	fbFeedback 			: FB_XP_Feedback(ipSourceInfo := fbSourceInfo);	
	{attribute 'hide'}                   	
	eActiveCommand 		: CHALET_Nc.E_NcAxisCommands := CHALET_Nc.E_NcAxisCommands.None;

END_VAR


// Planar-Feedback objects
VAR
	{attribute 'hide'} 
	fbFeedbackDisable : MC_PlanarFeedback;
	{attribute 'hide'} 
	fbFeedbackEnable : MC_PlanarFeedback;
	{attribute 'hide'} 
	fbFeedbackReset : MC_PlanarFeedback;
END_VAR

METHOD AddEnvironment : HRESULT
VAR_INPUT
	refEnvironment : REFERENCE TO MC_PlanarEnvironment;
	refFeedback : REFERENCE TO MC_PlanarFeedback;
END_VAR
refEnvironment.AddToGroup(refFeedback, fbGroup);
END_METHOD

METHOD AddMover : HRESULT
VAR_INPUT
	refMover : REFERENCE TO MC_PlanarMover;
	refFeedback : REFERENCE TO MC_PlanarFeedback;
END_VAR
refMover.AddToGroup(refFeedback, fbGroup);
END_METHOD

METHOD AddTrack : HRESULT
VAR_INPUT
	refTrack : REFERENCE TO MC_PlanarTrack;
	refFeedback : REFERENCE TO MC_PlanarFeedback;
END_VAR
refTrack.AddToGroup(refFeedback, fbGroup);
END_METHOD

METHOD Disable : HRESULT
VAR_INPUT
END_VAR
THIS^.eActiveCommand 				:= CHALET_NC.E_NcAxisCommands.Disable;
THIS^.fbFeedback.ActiveCommand 		:= TO_STRING(THIS^.eActiveCommand);	
THIS^.fbFeedback.LastCommandAccepted:= TRUE;		
THIS^.fbFeedback.Busy 				:= TRUE;

THIS^.fbGroup.Disable(fbFeedbackDisable);

Disable := S_OK;
END_METHOD

METHOD Enable : HRESULT
VAR_INPUT
END_VAR
IF NOT THIS^.fbFeedback.Busy THEN
	THIS^.eActiveCommand 				:= CHALET_NC.E_NcAxisCommands.Enable;
	THIS^.fbFeedback.ActiveCommand 		:= TO_STRING(THIS^.eActiveCommand);	
	THIS^.fbFeedback.LastCommandAccepted:= TRUE;		
	THIS^.fbFeedback.Busy 				:= TRUE;

	THIS^.fbGroup.Enable(fbFeedbackEnable);
	Enable := S_OK;
ELSE
	Enable := S_FALSE;
	THIS^.fbFeedback.LastCommandAccepted:= FALSE;	
END_IF
END_METHOD

METHOD FB_init : BOOL
VAR_INPUT
	bInitRetains : BOOL; // if TRUE, the retain variables are initialized (warm start / cold start)
	bInCopyCode : BOOL;  // if TRUE, the instance afterwards gets moved into the copy code (online change)
	
	ipSystem : I_CH_Object;
END_VAR
//Do the following code once during start up and not during onlinechange
IF NOT bInCopyCode THEN 
	

	(* Register to the Xplanar System
	   1. Test if the interface exists
	   2. Test if the object implements a "System for Mover" interface 
	*)
	IF ipSystem <> 0 AND_THEN __QUERYINTERFACE(ipSystem,THIS^.ipXpSystem) THEN
		THIS^.ipXpSystem.LinkGroup(THIS^);
	END_IF
	
	
	THIS^.fbFeedback.ActiveCommand 		:= TO_STRING(THIS^.eActiveCommand);	
	
END_IF
END_METHOD

{attribute 'monitoring':='call'}
PROPERTY Feedback : I_XP_Feedback
GET
Feedback := THIS^.fbFeedback;
END_GET
END_PROPERTY

METHOD Initialize : HRESULT
VAR_INPUT
END_VAR
VAR
	stVarInfo : __SYSTEM.VAR_INFO;
END_VAR
VAR_INST
	//This error cannot be reset. Requires a reset cold
	{attribute 'hide'}	
	fbInitError : FB_TcAlarm;
END_VAR
// Check if link to MC-Mover is mapped
IF NOT THIS^.Mapped THEN
	IF NOT fbInitError.bRaised THEN 
		//This error cannot be reset. Requires a reset cold
		fbInitError.CreateEx(stEventEntry:=TC_EVENTS.CHALET_Base_Events.VariableLinkMissing, ipSourceInfo := THIS^.fbSourceInfo, bWithConfirmation := FALSE);
		stVarInfo := __VARINFO(fbGroup);
		fbInitError.ipArguments.AddString(stVarInfo.Symbol);
		fbInitError.Raise(0);
	END_IF
	Initialize := E_FAIL;
	RETURN;
END_IF


IF NOT bInitDone THEN
	//Busy
	Initialize := S_PENDING;

	bInitDone := TRUE;	
	
ELSE	
	//Done
	Initialize := S_OK;	
END_IF


THIS^.eActiveCommand 				:= CHALET_NC.E_NcAxisCommands.Initialize;
THIS^.fbFeedback.ActiveCommand 		:= TO_STRING(THIS^.eActiveCommand);	
THIS^.fbFeedback.LastCommandAccepted:= TRUE;	
//Set done or keep in busy state	
THIS^.fbFeedback.HR := Initialize;
END_METHOD

{attribute 'monitoring':='call'}
PROPERTY Mapped : BOOL //Project is mapped to MC (McToPlc and PlcToMc)
GET
VAR
	bMcToPlcNotMapped 	: BOOL;
END_VAR
bMcToPlcNotMapped := F_GetMappingStatus(ADR(THIS^.fbGroup.MCTOPLC_STD), SIZEOF(THIS^.fbGroup.MCTOPLC_STD)) <> EPlcMappingStatus.MS_Mapped;

Mapped := NOT bMcToPlcNotMapped;
END_GET
END_PROPERTY

{attribute 'monitoring':='call'}
//Unique object ID
PROPERTY OID : OTCID
GET
OID := THIS^.fbGroup.MCTOPLC_STD.GroupOID;
END_GET
END_PROPERTY

{attribute 'monitoring':='call'}
PROPERTY PlanarGroup : REFERENCE TO MC_PlanarGroup
GET
PlanarGroup ref= THIS^.fbGroup;
END_GET
END_PROPERTY

METHOD Reset : HRESULT
VAR_INPUT
END_VAR
IF NOT THIS^.fbFeedback.Busy THEN
	THIS^.eActiveCommand 				:= CHALET_NC.E_NcAxisCommands.Reset;
	THIS^.fbFeedback.ActiveCommand 		:= TO_STRING(THIS^.eActiveCommand);	
	THIS^.fbFeedback.LastCommandAccepted:= TRUE;		
	THIS^.fbFeedback.Busy 				:= TRUE;

	THIS^.fbGroup.Reset(fbFeedbackReset);
	Reset := S_OK;
ELSE
	Reset := S_FALSE;
	THIS^.fbFeedback.LastCommandAccepted:= FALSE;		
END_IF
END_METHOD

{attribute 'monitoring':='call'}
//Interface to CHALET system to which this object belongs
PROPERTY System : I_XP_System_PLC
GET
//get I_x_System_PLC interface from I_x_System_Registration
__QUERYINTERFACE(THIS^.ipXpSystem, System);
END_GET
END_PROPERTY

METHOD PUBLIC Update : HRESULT
VAR_INPUT
END_VAR



// ********************** Set feedback depending on active command *******************************
CASE THIS^.eActiveCommand OF
	E_NcAxisCommands.None: 
		//Display if a Mover Error is active during no command is active
		IF THIS^.fbGroup.Error AND NOT fbFeedback.Error THEN 
			fbFeedback.ErrorId 			:= THIS^.fbGroup.ErrorID;
			fbFeedback.ActiveCommand 	:= TO_STRING(E_NcAxisCommands.None);	
			fbFeedback.ClearObjectInfo();
		END_IF

	E_NcAxisCommands.Initialize:
		fbFeedback.Busy 			:= NOT THIS^.bInitDone;
		fbFeedback.Done 			:= THIS^.bInitDone;
		fbFeedback.ErrorId 			:= 0;
		fbFeedback.ClearObjectInfo();
		                        	
	E_NcAxisCommands.Enable:     	
		fbFeedback.Busy 			:= fbFeedbackEnable.Busy;
		fbFeedback.Done 			:= fbFeedbackEnable.Done;
		fbFeedback.ErrorId 			:= fbFeedbackEnable.ErrorID;
        fbFeedback.ObjectInfo		:= fbFeedbackEnable.objectInfo;
                                			                        	
	E_NcAxisCommands.Disable:     	
		fbFeedback.Busy 			:= fbFeedbackDisable.Busy;
		fbFeedback.Done 			:= fbFeedbackDisable.Done;
		fbFeedback.ErrorId 			:= fbFeedbackDisable.ErrorID;
        fbFeedback.ObjectInfo		:= fbFeedbackDisable.objectInfo;
                                			                        	
	E_NcAxisCommands.Reset:     	
		fbFeedback.Busy 			:= fbFeedbackReset.Busy;
		fbFeedback.Done 			:= fbFeedbackReset.Done;
		fbFeedback.ErrorId 			:= fbFeedbackReset.ErrorID;
        fbFeedback.ObjectInfo		:= fbFeedbackReset.objectInfo;
                                		
	ELSE//External command in subclass
		;
END_CASE


// **********************  Stop to execute commands on .done or .error ***************************
IF fbFeedback.Done OR THIS^.fbFeedback.Error THEN
	eActiveCommand 				:= E_NcAxisCommands.None;
END_IF

//Update xplanar object
THIS^.fbGroup.Update();

//Update feedback object
fbFeedbackEnable.Update(); 
fbFeedbackDisable.Update(); 
fbFeedbackReset.Update();
END_METHOD

END_FUNCTION_BLOCK

// ---- COMPONENTs/System/FB_XP_System.TcPOU
{attribute 'no_explicit_call' := 'Do not call the body - Stick to OOP'}
(* XPlanar System - 1 per associated XPlanar 
	The system is the container and organizer for all subsequent XPlanar objects. All objects are registered with this system*)
FUNCTION_BLOCK FB_XP_System EXTENDS FB_CH_Object IMPLEMENTS I_XP_System_Registration, I_XP_System_PLC
VAR	
	{attribute 'hide'}
	bInitDone : BOOL;
	{attribute 'hide'}
	bErrorDuringFbInit : BOOL; // Not possible to reset
	{attribute 'hide'}                   	
	eActiveCommand 		: CHALET_Nc.E_NcAxisCommands := CHALET_Nc.E_NcAxisCommands.None;
	{attribute 'hide'}
    fbMoversPresent     : FB_CH_List;
	{attribute 'hide'}
    fbMoversNotPresent 	: FB_CH_List;
	{attribute 'hide'}
	fbListAllMovers 	: FB_CH_List;
	{attribute 'hide'}	
    fbTracks    		: FB_CH_List;
	{attribute 'hide'}	
	fbStationsAll 	 : FB_CH_List;//List of all station objects that exist in this project
	{attribute 'hide'}	
	fbStationsUsed 	 : FB_CH_List;//List of all station objects that are considered for path planning in the currently running system
	{attribute 'hide'}	
	fbTriggers 	 : FB_CH_List;
	{attribute 'hide'}	
	fbZones 	 : FB_CH_List;
	{attribute 'hide'}	
	fbPaths 	 : FB_CH_List;
	{attribute 'hide'}	
    ipGroup       : I_XP_Group;
	{attribute 'hide'}	
    ipEnvironment : I_XP_Environment;
	{attribute 'hide'}
    nSeqEnabling  : UINT;
	{attribute 'hide'}
	nSeqJoiningTrack : UINT;
	{attribute 'hide'}
	nSeqJoiningStation : UINT;
	{attribute 'hide'}	
    nSeqDisabling  : UINT := SEQ_DONE;
	{attribute 'hide'}
	fbFeedback : FB_CH_Feedback(ipSourceInfo := fbSourceInfo);	
END_VAR
VAR CONSTANT
	{attribute 'hide'}
	SEQ_DONE : UINT := 999;
END_VAR

METHOD AddMoverToSystem : HRESULT
VAR_INPUT
	ipMover : I_XP_Mover;
	xPos, yPos : LREAL;
END_VAR
VAR
	stParameter : EnterOrLeaveMovementAreaParameters;
END_VAR
IF ipMover <> 0 THEN
	THIS^.fbMoversNotPresent.RemoveObject(ipMover);
	
	//Add if not already in list
	IF NOT THIS^.fbMoversPresent.ObjectInList(ipMover) THEN
		THIS^.fbMoversPresent.AddObject(ipMover);
	END_IF
	
	//todo
//	stParameter.
//	ipMover.TcIoXPlanarMover.SetMovementArea(stParameter);
END_IF
END_METHOD

METHOD CheckForErrors : BOOL
VAR
	ipEachMover : I_XP_Mover;
	bErrorFound : BOOL;
	bAtLeastOnMoverIsEnabled : BOOL;
END_VAR
VAR_INST
	{attribute 'hide'}
	bErrorFoundOld : BOOL;
END_VAR
THIS^.fbMoversPresent.ResetIterator();
WHILE THIS^.fbMoversPresent.HasNextObject() DO
	IF __QUERYINTERFACE(THIS^.fbMoversPresent.GetNextObject(),ipEachMover) THEN
			bErrorFound := bErrorFound OR ipEachMover.Feedback.Error;
			bErrorFound := bErrorFound OR (ipEachMover.PlanarMover.MCTOPLC.STD.ErrorCode <> 0);
									
			//Only Disable System on Error, if at least on Mover is Enabled
			bAtLeastOnMoverIsEnabled := ipEachMover.Enabled OR bAtLeastOnMoverIsEnabled;
	END_IF
END_WHILE
THIS^.fbMoversPresent.RestoreIterator();

//check this system (Enabling disabling)
bErrorFound := bErrorFound OR THIS^.fbFeedback.Error;


//Do an disable at new error found
IF bAtLeastOnMoverIsEnabled AND bErrorFound AND NOT bErrorFoundOld THEN 
	THIS^.Disable();
END_IF

//Keep information
bErrorFoundOld := bErrorFound;
END_METHOD

METHOD CheckTargetExists : BOOL //Return TRUE if target is existing
VAR_INPUT
	sStation	: STRING; //Group of the target station or LUID
END_VAR
VAR
	ipEachStation : I_XP_Station_PLC;
END_VAR
THIS^.fbStationsUsed.ResetIterator();
WHILE THIS^.fbStationsUsed.HasNextObject() DO
	IF __QUERYINTERFACE(THIS^.fbStationsUsed.GetNextObject(),ipEachStation) THEN
		//Return TRUE if found
		IF (ipEachStation.TargetGroupe = sStation) OR (ipEachStation.LUID = sStation) THEN
			CheckTargetExists := TRUE;
			EXIT;
		END_IF
	END_IF
END_WHILE
THIS^.fbStationsUsed.RestoreIterator();
END_METHOD

METHOD PROTECTED CreateHelpStations : HRESULT
VAR

END_VAR
VAR_INST
	{attribute 'hide'}	
	fbDelayJoiningStation : TON;
END_VAR
CASE nSeqCreateHelpStations OF

	0: //Init
		fbDelayJoiningStation.IN := FALSE;
		nSeqJoiningStation := 10;
	
	
		
		IF CheckOk(hr) THEN 
			nSeqJoiningStation := SEQ_DONE;
		ELSIF FAILED(hr) THEN
			nSeqJoiningStation := 1000 + nSeqJoiningStation;
		END_IF			

	
	1000..1999://Error
		hr := GetMostSignificant(hr, E_FAIL);
END_CASE



//Return value
IF FAILED(hr) THEN 
	//Error
    CreateHelpStations := GetMostSignificant(hr, E_FAIL);
ELSIF (nSeqCreateHelpStations = SEQ_DONE) THEN
	//Done
    CreateHelpStations := S_OK;
ELSE
	//Busy
    CreateHelpStations := S_PENDING;;
END_IF
END_METHOD

METHOD Disable : I_CH_Feedback
VAR_INPUT
END_VAR
//Disable is allways posible, but only if not already active
IF THIS^.nSeqDisabling = 0 OR THIS^.nSeqDisabling >= SEQ_DONE THEN
	THIS^.nSeqDisabling 	:= 1;
	THIS^.nSeqEnabling 		:= 0;
	
	THIS^.eActiveCommand 					:= CHALET_NC.E_NcAxisCommands.Disable;
	THIS^.fbFeedback.ActiveCommand 			:= TO_STRING(THIS^.eActiveCommand);	
	THIS^.fbFeedback.LastCommandAccepted	:= TRUE;		
	THIS^.fbFeedback.Busy 					:= TRUE;
			
	
ELSE
	THIS^.fbFeedback.LastCommandAccepted	:= FALSE;	
END_IF

Disable := THIS^.fbFeedback;
END_METHOD

{attribute 'monitoring':='call'}
PROPERTY Disabled : BOOL
GET
Disabled := nSeqDisabling = SEQ_DONE OR 
			(nSeqDisabling = 0 AND nSeqEnabling = 0);
END_GET
END_PROPERTY

METHOD PROTECTED Disabling : HRESULT
VAR
	hr : HRESULT;
	bOk : BOOL := TRUE;
	ipEachMover : I_XP_Mover;
	ipEachTrack : I_XP_Track;
	ipEachStation : I_XP_Station;
END_VAR
VAR_INST
	hrLastCycle : HRESULT;
END_VAR
Disabling := S_PENDING;
CASE nSeqDisabling OF
	0: // Idle
		Disabling := S_OK;
		
		
	1: // Halt movers - keep at first position for a fast stop reaction
		THIS^.fbMoversPresent.ResetIterator();
		WHILE THIS^.fbMoversPresent.HasNextObject() DO
			IF ToXpMover(THIS^.fbMoversPresent.GetNextObject(),ipEachMover) THEN
				IF XPlanarParameterlist.B_QUICKSTOP_ON_DISABLING THEN
					//The mover stops immediately at the current position
					hr := GetMostSignificant(hr, ipEachMover.Disable());
				ELSE
					//The mover cancels the superimposed ExternalSetpoint movement and returns to the track with maximum dynamic. -> Like a rubber band
					hr := GetMostSignificant(hr, ipEachMover.Halt());
				END_IF
			END_IF
		END_WHILE
		THIS^.fbMoversPresent.RestoreIterator();
	    		
		IF CheckOk(hr) THEN 
			nSeqDisabling := 20;
		ELSE
			nSeqDisabling := 1000 + nSeqDisabling;
		END_IF	
	
		
	20: // Halting movers
		THIS^.fbMoversPresent.ResetIterator();
		WHILE THIS^.fbMoversPresent.HasNextObject() DO
			IF ToXpMover(THIS^.fbMoversPresent.GetNextObject(),ipEachMover) THEN
				bOk := bOk AND ipEachMover.Standstill;
			END_IF
		END_WHILE
		THIS^.fbMoversPresent.RestoreIterator();
		
		IF bOk THEN 
			nSeqDisabling := 30;
		END_IF	
			
		
	
	30: // Reset movers
		THIS^.fbMoversPresent.ResetIterator();
		WHILE THIS^.fbMoversPresent.HasNextObject() DO
			IF ToXpMover(THIS^.fbMoversPresent.GetNextObject(),ipEachMover) THEN
				hr := GetMostSignificant(hr, ipEachMover.Reset());
			END_IF
		END_WHILE
		
		IF CheckOk(hr) THEN 
			nSeqDisabling := 40;
		ELSE
			nSeqDisabling := 1000 + nSeqDisabling;
		END_IF		
		
		
	40: // Resetting movers
		THIS^.fbMoversPresent.ResetIterator();
		WHILE THIS^.fbMoversPresent.HasNextObject() DO
			IF ToXpMover(THIS^.fbMoversPresent.GetNextObject(),ipEachMover) THEN
				hr := GetMostSignificant(hr, ipEachMover.Feedback.HR);
			END_IF
		END_WHILE
		
		IF CheckOk(hr) THEN 
		//	nSeqDisabling := 45;
			nSeqDisabling := 50;
		ELSIF FAILED(hr) THEN
			nSeqDisabling := 1000 + nSeqDisabling;
		END_IF
		
		
		
(*		
	45: // Stop external Setpoint 
		THIS^.fbMovers.ResetIterator();
		WHILE THIS^.fbMovers.HasNextObject() DO
			IF ToXpMover(THIS^.fbMovers.GetNextObject(),iTempMover) THEN
				hr := GetMostSignificant(hr, iTempMover.StopExternalSetpoint());
			END_IF
		END_WHILE
		
		IF CheckOk(hr) THEN 
			nSeqDisabling := 46;
		ELSE
			nSeqDisabling := 1000 + nSeqDisabling;
		END_IF			
		

	46: // Stoping external Setpoint 
		THIS^.fbMovers.ResetIterator();
		WHILE THIS^.fbMovers.HasNextObject() DO
			IF ToXpMover(THIS^.fbMovers.GetNextObject(),iTempMover) THEN
				hr := GetMostSignificant(hr, iTempMover.Feedback.HR);
			END_IF
		END_WHILE
		
		IF CheckOk(hr) THEN 
			nSeqDisabling := 50;
		ELSIF FAILED(hr) THEN
			nSeqDisabling := 1000 + nSeqDisabling;
		END_IF			
*)		
		
		
		
	50: // Disable movers
		THIS^.fbMoversPresent.ResetIterator();
		WHILE THIS^.fbMoversPresent.HasNextObject() DO
			IF ToXpMover(THIS^.fbMoversPresent.GetNextObject(),ipEachMover) THEN
				hr := GetMostSignificant(hr, ipEachMover.Disable());
			END_IF
		END_WHILE
		
		IF CheckOk(hr) THEN 
			nSeqDisabling := 60;
		ELSE
			nSeqDisabling := 1000 + nSeqDisabling;
		END_IF			
		

		
	60: // Disabling movers
		THIS^.fbMoversPresent.ResetIterator();
		WHILE THIS^.fbMoversPresent.HasNextObject() DO
			IF ToXpMover(THIS^.fbMoversPresent.GetNextObject(),ipEachMover) THEN
				hr := GetMostSignificant(hr, ipEachMover.Feedback.HR);
			END_IF
		END_WHILE
		
		IF CheckOk(hr) THEN 
			nSeqDisabling := 61;
		ELSIF FAILED(hr) THEN
			nSeqDisabling := 1000 + nSeqDisabling;
		END_IF		


	61: // Reset track
		THIS^.fbTracks.ResetIterator();
		WHILE THIS^.fbTracks.HasNextObject() DO
			IF ToXpTrack(THIS^.fbTracks.GetNextObject(),ipEachTrack) THEN
				hr := GetMostSignificant(hr, ipEachTrack.Reset());
			END_IF
		END_WHILE
		
		IF CheckOk(hr) THEN 
			nSeqDisabling := 62;
		ELSE
			nSeqDisabling := 1000 + nSeqDisabling;
		END_IF		
		
		
	62: // Resetting track
		THIS^.fbTracks.ResetIterator();
		WHILE THIS^.fbTracks.HasNextObject() DO
			IF ToXpTrack(THIS^.fbTracks.GetNextObject(),ipEachTrack) THEN
				hr := GetMostSignificant(hr, ipEachTrack.Feedback.HR);
			END_IF
		END_WHILE
		
		IF CheckOk(hr) THEN 
			nSeqDisabling := 63;
		ELSIF FAILED(hr) THEN
			nSeqDisabling := 1000 + nSeqDisabling;
		END_IF	

				
	63: // Reset group
		hr := ipGroup.Reset();
		
		IF CheckOk(hr) THEN 
			nSeqDisabling := 64;
		ELSE
			nSeqDisabling := 1000 + nSeqDisabling;
		END_IF		
		
		
	64: // Resetting group
		hr := ipGroup.Feedback.HR;
		
		IF CheckOk(hr) THEN 
			nSeqDisabling := 70;
		ELSIF FAILED(hr) THEN
			nSeqDisabling := 1000 + nSeqDisabling;
		END_IF		
		
		
		

   70: // Disable tracks
		THIS^.fbTracks.ResetIterator();
		WHILE THIS^.fbTracks.HasNextObject() DO
			IF ToXpTrack(THIS^.fbTracks.GetNextObject(),ipEachTrack) THEN
				hr := GetMostSignificant(hr, ipEachTrack.Disable());
			END_IF
		END_WHILE
		
		IF CheckOk(hr) THEN 
			nSeqDisabling := 80;
		ELSE
			nSeqDisabling := 1000 + nSeqDisabling;
		END_IF			
   
		
   80: // Disabling tracks
		THIS^.fbTracks.ResetIterator();
		WHILE THIS^.fbTracks.HasNextObject() DO
			IF ToXpTrack(THIS^.fbTracks.GetNextObject(),ipEachTrack) THEN
				hr := GetMostSignificant(hr, ipEachTrack.Feedback.HR);
			END_IF
		END_WHILE
		
		IF CheckOk(hr) THEN 
			nSeqDisabling := 90;
		ELSIF FAILED(hr) THEN
			nSeqDisabling := 1000 + nSeqDisabling;
		END_IF	
				

	90: // Disable group
		hr := ipGroup.Disable();
		
		IF CheckOk(hr) THEN 
			nSeqDisabling := 100;
		ELSE
			nSeqDisabling := 1000 + nSeqDisabling;
		END_IF	
		
		
   100: // Disabling group
		hr := ipGroup.Feedback.HR;
		
		IF CheckOk(hr) THEN 
			nSeqDisabling := 102;
		ELSIF FAILED(hr) THEN
			nSeqDisabling := 1000 + nSeqDisabling;
		END_IF	

		
	102: //Delete all paths. These are only temporary objects and will be recreated the next time they are enabled
		THIS^.fbStationsUsed.ResetIterator();
		WHILE THIS^.fbStationsUsed.HasNextObject() DO
			IF ToXpStation(THIS^.fbStationsUsed.GetNextObject(),ipEachStation) THEN
				hr := ipEachStation.Disassemble();
			END_IF
		END_WHILE
	
		IF CheckOk(hr) THEN 
			nSeqDisabling := 103;
		ELSE
			nSeqDisabling := 1000 + nSeqDisabling;
		END_IF			
		
		
	103: //Delete all paths. These are only temporary objects and will be recreated the next time they are enabled
		THIS^.fbListAllMovers.ResetIterator();
		WHILE THIS^.fbListAllMovers.HasNextObject() DO
			IF ToXpMover(THIS^.fbListAllMovers.GetNextObject(),ipEachMover) THEN
				hr := ipEachMover.Disassemble();
			END_IF
		END_WHILE
	
		IF CheckOk(hr) THEN 
			nSeqDisabling := 105;
		ELSE
			nSeqDisabling := 1000 + nSeqDisabling;
		END_IF		
		
		
		
		
		
  105: // Remove tracks from group
		THIS^.fbTracks.ResetIterator();
		WHILE THIS^.fbTracks.HasNextObject() DO
			IF ToXpTrack(THIS^.fbTracks.GetNextObject(),ipEachTrack) THEN
				hr := GetMostSignificant(hr, ipEachTrack.RemoveFromGroup());
			END_IF
		END_WHILE
		
		IF CheckOk(hr) THEN 
			nSeqDisabling := 106;
		ELSE
			nSeqDisabling := 1000 + nSeqDisabling;
		END_IF			
   
		
   106: // Removing tracks from group
		THIS^.fbTracks.ResetIterator();
		WHILE THIS^.fbTracks.HasNextObject() DO
			IF ToXpTrack(THIS^.fbTracks.GetNextObject(),ipEachTrack) THEN
				bOk := bOk AND ipEachTrack.PlanarTrack.MCTOPLC_STD.GroupOID = 0;
			END_IF
		END_WHILE
		
		IF bOk THEN 
			nSeqDisabling := 110;
		END_IF	
		
		
	110: // Remove movers from group
		THIS^.fbMoversPresent.ResetIterator();
		WHILE THIS^.fbMoversPresent.HasNextObject() DO
			IF ToXpMover(THIS^.fbMoversPresent.GetNextObject(),ipEachMover) THEN
				hr := GetMostSignificant(hr, ipEachMover.RemoveFromGroup());
			END_IF
		END_WHILE
		
		IF CheckOk(hr) THEN 
			nSeqDisabling := 120;
		ELSE
			nSeqDisabling := 1000 + nSeqDisabling;
		END_IF		
	
		
	120: // Removing movers from group
		THIS^.fbMoversPresent.ResetIterator();
		WHILE THIS^.fbMoversPresent.HasNextObject() DO
			IF ToXpMover(THIS^.fbMoversPresent.GetNextObject(),ipEachMover) THEN
				bOk := bOk AND ipEachMover.PlanarMover.MCTOPLC.STD.GroupOID = 0;
			END_IF
		END_WHILE
		
		IF bOk THEN 
			nSeqDisabling := 130;
		END_IF		
	
		
	130: // Remove envirement from group
		hr := ipEnvironment.RemoveFromGroup();
		
		IF CheckOk(hr) THEN 
			nSeqDisabling := 140;
		ELSE
			nSeqDisabling := 1000 + nSeqDisabling;
		END_IF		
		
		
   140: // Removing envirement from group
		hr := ipEnvironment.Feedback.HR;
	
		IF CheckOk(hr) THEN 
			nSeqDisabling := 200;
		ELSIF FAILED(hr) THEN
			nSeqDisabling := 1000 + nSeqDisabling;
		END_IF			
		
		
   200: // Reset Utility errors
		ipEnvironment.UtilityEnvirement.ErrorAcknowledge();
		nSeqDisabling := SEQ_DONE;

		
	
   SEQ_DONE: //Done
   		Disabling := S_OK;

		
	1000..1999://Error
		hr := GetMostSignificant(hrLastCycle, E_FAIL);
	
END_CASE

//store last information
hrLastCycle := hr;

// Propagate error
IF FAILED(hr) THEN
	Disabling := hr;
END_IF
END_METHOD

METHOD Enable : CHALET_BaseComponents.I_CH_Feedback
VAR_INPUT
END_VAR
IF NOT THIS^.fbFeedback.Done THEN
	//Error active/not ready
	THIS^.fbFeedback.LastCommandAccepted 	:= FALSE;

ELSIF nSeqEnabling <> 0 THEN
	//System is partial or full enabled. Disable first.
	THIS^.fbFeedback.LastCommandAccepted 	:= FALSE;
ELSE
	THIS^.nSeqDisabling 	:= 0;
	THIS^.nSeqEnabling 		:= 1;
	
	THIS^.eActiveCommand 				:= CHALET_NC.E_NcAxisCommands.Enable;
	THIS^.fbFeedback.ActiveCommand 		:= TO_STRING(THIS^.eActiveCommand);	
	THIS^.fbFeedback.LastCommandAccepted:= TRUE;		
	THIS^.fbFeedback.Busy 				:= TRUE;	
END_IF

Enable := THIS^.fbFeedback;
END_METHOD

{attribute 'monitoring':='call'}
PROPERTY Enabled : BOOL
GET
Enabled := nSeqEnabling = SEQ_DONE;
END_GET
END_PROPERTY

METHOD PROTECTED Enabling : HRESULT
VAR

	hr : HRESULT;
	bWatchDogActive : BOOL;
	ipTempMover : I_XP_Mover;
	ipTempMoverPlc : I_XP_Mover_PLC;
	ipTempStation : I_XP_Station;
	ipTempTrack : I_XP_Track;
	stController : ST_TcIoControllersOn;
	lrCRotationShortestPos : LREAL;
	bOk : BOOL;
	nSupSeq : UINT;
	nIdx : UINT;
	sMoverType : STRING;
	fDistLastToSet : LREAL;
	fMaxError : LREAL;
	nMoversDetected, nMoverExpected : UDINT;
	bMoverIsMissing : BOOL;
	eMoverDetectionStatus : MoverDetectionStatus;
	stCoordMoverCommStatus : CoordinatedMoverCommStatus;
	ipMoverTComObject : ITComObject;
	nParaSize : UDINT;
	pParaData : PVOID;
	eAccessory : MoverAccessoryID;//(APM9000_0000:=0, APM9001_0000:=1)
END_VAR

VAR_INST
	{attribute 'hide'}	
	fbTimeOutSeq : TON; 
	{attribute 'hide'}	
	hrLastCycle 	: HRESULT;
	{attribute 'hide'}	
	nlastState	: UINT;
	
	// todo hide
	bIdBumperOnAllMovers : BOOL;
	
	{attribute 'hide'}	
	fbTimeOutEnabling : FB_TcAlarm;
	{attribute 'hide'}	
	fbErrorEnabling : FB_TcAlarm;
	{attribute 'hide'}	
	fbErrorMoverDetection : FB_TcAlarm;
	{attribute 'hide'}	
	bAllMoverOrientationValide : BOOL;	
	{attribute 'hide'}	
	bAllMoverIdDetectionValide : BOOL;
END_VAR
Enabling := S_PENDING;
CASE nSeqEnabling OF
	0: // Idle
		Enabling := S_OK;	
				
	1: // Prepare 
		THIS^.fbListAllMovers.Clear();
		THIS^.fbListAllMovers.AddList(THIS^.fbMoversPresent);
		THIS^.fbListAllMovers.AddList(THIS^.fbMoversNotPresent);
		
		
		////Are ID-Bumpers configured on each mover?
		//bIdBumperOnAllMovers := TRUE;
		//THIS^.fbListAllMovers.ResetIterator();
		//WHILE THIS^.fbListAllMovers.HasNextObject() DO
		//	IF ToXpMover(THIS^.fbListAllMovers.GetNextObject(),ipTempMover) THEN
		//		eAccessory := ipTempMover.TcIoXPlanarMover.GetAccessoryId(1);
		//		bIdBumperOnAllMovers := bIdBumperOnAllMovers AND (eAccessory = MoverAccessoryID.APM9001_0000);
		//	END_IF
		//END_WHILE
		//Todo: Read of GetAccessoryId will crash the system if mover is not present
		bIdBumperOnAllMovers := XPlanarParameterlist.B_ID_BUMPER_INSTALLED;
		
		IF (THIS^.ipEnvironment.UtilityEnvirement.TcIoXpu(1).GetOperationMode() = XplanarOperationMode.Normal) THEN
			// Hardware - Do detection
			nSeqEnabling := 4;
		ELSE
			// Simulation - Skip detection
			nSeqEnabling := 20;
		END_IF


	4: //Redetect all movers on real system
		//timeout is monitored in this sequence
		bWatchDogActive := TRUE;

		//check if all mover are present
		THIS^.fbMoversPresent.ResetIterator();
		WHILE THIS^.fbMoversPresent.HasNextObject() DO
			IF ToXpMover(THIS^.fbMoversPresent.GetNextObject(),ipTempMover) AND_THEN ipTempMover.MoverIsNotPresent THEN
				bMoverIsMissing := TRUE;
				bAllMoverOrientationValide := FALSE;
				bAllMoverIdDetectionValide := FALSE;
			END_IF
		END_WHILE
		THIS^.fbMoversPresent.RestoreIterator();
				
		//Decidif no ID-Bmper is installed, it is better not to do an unnecessary redetect, as the movers renumber themselves. 
		//If an ID bumper is present, a detection can be made without any problems whether a mover detection should be made or not
		// - However, as this takes a very long time, it is dispensed with
		IF bMoverIsMissing (*OR bIdBumperOnAllMovers*) THEN
			THIS^.ipEnvironment.UtilityEnvirement.TcIoXpu(1).SetStartMoverRedetection();
			nSeqEnabling := 5;
		ELSE
			//skip redetection
			nSeqEnabling := 6;
		END_IF

	5: //Wait for finish redetection
		//timeout is monitored in this sequence
		bWatchDogActive := TRUE;
		eMoverDetectionStatus := THIS^.Enviroment.ProcessingUnitMoverDetectionStatus;
		IF (eMoverDetectionStatus = MoverDetectionStatus.DetectionSuccessful) THEN
			nSeqEnabling := 6;
		END_IF

		
	6: //Compare detectet and expectet movers	
	   //timeout is monitored in this sequence
		bWatchDogActive := TRUE;
		nSeqEnabling := 10;	
		
		//Todo error if mover is missing
//		FOR nIdx := 0 TO 5 DO
//			CASE nIdx OF
//				0:  sMoverType		:= 'APM4220';
//					nMoverExpected 	:= THIS^.ipEnvironment.UtilityEnvirement.TcIoXpu(1).GetMoverDetectionInfos().APM4220Expected;
//					nMoversDetected := THIS^.ipEnvironment.UtilityEnvirement.TcIoXpu(1).GetMoverDetectionInfos().APM4220Detected;
//				1: 	sMoverType		:= 'APM4221';
//					nMoverExpected 	:= THIS^.ipEnvironment.UtilityEnvirement.TcIoXpu(1).GetMoverDetectionInfos().APM4221Expected;
//					nMoversDetected := THIS^.ipEnvironment.UtilityEnvirement.TcIoXpu(1).GetMoverDetectionInfos().APM4221Detected;
//				2:  sMoverType		:= 'APM4330';
//					nMoverExpected 	:= THIS^.ipEnvironment.UtilityEnvirement.TcIoXpu(1).GetMoverDetectionInfos().APM4330Expected;
//					nMoversDetected := THIS^.ipEnvironment.UtilityEnvirement.TcIoXpu(1).GetMoverDetectionInfos().APM4330Detected;
//				3:  sMoverType		:= 'APM4550';
//					nMoverExpected 	:= THIS^.ipEnvironment.UtilityEnvirement.TcIoXpu(1).GetMoverDetectionInfos().APM4550Expected;
//					nMoversDetected := THIS^.ipEnvironment.UtilityEnvirement.TcIoXpu(1).GetMoverDetectionInfos().APM4550Detected;
//				4:  sMoverType		:= 'total mover count';
//					nMoverExpected 	:= THIS^.ipEnvironment.UtilityEnvirement.TcIoXpu(1).GetMoverDetectionInfos().TotalExpected;
//					nMoversDetected := THIS^.ipEnvironment.UtilityEnvirement.TcIoXpu(1).GetMoverDetectionInfos().TotalDetected;
//					
//				5: //Succesfull finished
//					nSeqEnabling := 10;	
//			END_CASE	
//
//			IF nMoverExpected <> nMoversDetected THEN
//				//Error
//				nSeqEnabling := 1000 + nSeqEnabling;
//				fbErrorMoverDetection.CreateEx(stEventEntry:=TC_EVENTS.CHALET_XPlanar_Events.MoverDetectionFailed, ipSourceInfo := THIS^.fbSourceInfo, bWithConfirmation := FALSE);
//				//Mover detection failed. Expected {0} found {1} of type {2}
//				fbErrorMoverDetection.ipArguments.AddUDInt(nMoverExpected).AddUDInt(nMoversDetected).AddStringByValue(sMoverType);
//				fbErrorMoverDetection.Raise(0);
//				EXIT;
//			END_IF		
//		END_FOR
		
	
	//ID
	10: //Deside if or if not to get ID of mover. Require an APM9001-0000-4xxx | XPlanar-ID-Bumper
		bWatchDogActive := TRUE;
		IF XPlanarParameterlist.B_GET_MOVER_ID AND bIdBumperOnAllMovers AND NOT bAllMoverIdDetectionValide THEN
			THIS^.ipEnvironment.UtilityEnvirement.TcIoXpu(1).SetCoordMoverCommunicationCmd(CoordinatedMoverCommCommand.IdentifyAndAssignPossible);
			nSeqEnabling := 11;
		ELSE
			nSeqEnabling := 15;
		END_IF		
		
	11: //Wait for start of comm
		bWatchDogActive := TRUE;
		stCoordMoverCommStatus :=  THIS^.ipEnvironment.UtilityEnvirement.TcIoXpu(1).GetCoordMoverCommStatus();
		IF stCoordMoverCommStatus = CoordinatedMoverCommStatus.CommunicationInProcess THEN
			nSeqEnabling := nSeqEnabling +1;
		END_IF	
		
	12: // Check result of mover identification
		bWatchDogActive := TRUE;
		stCoordMoverCommStatus :=  THIS^.ipEnvironment.UtilityEnvirement.TcIoXpu(1).GetCoordMoverCommStatus();
		IF stCoordMoverCommStatus = CoordinatedMoverCommStatus.CommunicationSuccessful THEN
			bAllMoverIdDetectionValide := TRUE;
			nSeqEnabling := 15;
		ELSIF stCoordMoverCommStatus = CoordinatedMoverCommStatus.CommunicationFailed THEN
			// Error: CommunicationFailed
			nSeqEnabling := 1000 + nSeqEnabling;
		END_IF
		
		
		
	//Orientation
	15://Deside if or if not to get orientation of mover. Require an APM9001-0000-4xxx | XPlanar-ID-Bumper
		bWatchDogActive := TRUE;
		IF XPlanarParameterlist.B_GET_MOVER_ORIENTATION AND bIdBumperOnAllMovers AND NOT bAllMoverOrientationValide THEN
			THIS^.ipEnvironment.UtilityEnvirement.TcIoXpu(1).SetCoordMoverCommunicationCmd(CoordinatedMoverCommCommand.DetermineOrientations);
			nSeqEnabling:= 16;
		ELSE
			nSeqEnabling := 20;
		END_IF	
	
	16: //Wait for start of comm
		bWatchDogActive := TRUE;
		stCoordMoverCommStatus :=  THIS^.ipEnvironment.UtilityEnvirement.TcIoXpu(1).GetCoordMoverCommStatus();
		IF stCoordMoverCommStatus = CoordinatedMoverCommStatus.CommunicationInProcess THEN
			nSeqEnabling := nSeqEnabling +1;
		END_IF		
		
	17: // Check result of mover orientation
		bWatchDogActive := TRUE;
		stCoordMoverCommStatus :=  THIS^.ipEnvironment.UtilityEnvirement.TcIoXpu(1).GetCoordMoverCommStatus();
		IF stCoordMoverCommStatus = CoordinatedMoverCommStatus.CommunicationSuccessful THEN
			nSeqEnabling := 20;
		ELSIF stCoordMoverCommStatus = CoordinatedMoverCommStatus.CommunicationFailed THEN
			// Error: CommunicationFailed
			nSeqEnabling := 1000 + nSeqEnabling;
		END_IF		
		
		
		
	20:	//Add movers in list present or not present
		IF XPlanarParameterlist.B_AUTOMATICALLY_REMOVE_NOT_PRESENT_MOVER_AT_ENABLING THEN
			THIS^.fbMoversPresent.Clear();
			THIS^.fbMoversNotPresent.Clear();
			THIS^.fbListAllMovers.ResetIterator();
			WHILE THIS^.fbListAllMovers.HasNextObject() DO
				IF ToXpMover(THIS^.fbListAllMovers.GetNextObject(),ipTempMover) THEN
					IF  ipTempMover.MoverIsNotPresent THEN
						THIS^.fbMoversNotPresent.AddObject(ipTempMover);
					ELSE
						THIS^.fbMoversPresent.AddObject(ipTempMover);
					END_IF
				END_IF
			END_WHILE
			THIS^.fbListAllMovers.RestoreIterator();
		END_IF		
		nSeqEnabling := 21;			
			

		
	21:	//Enable all position controllers(XYZABC) in Mover-TcCOM
		stController.x := TRUE;stController.y := TRUE;stController.z := TRUE;
		stController.a := TRUE;stController.b := TRUE;stController.c := TRUE;
		THIS^.fbMoversPresent.ResetIterator();
		WHILE THIS^.fbMoversPresent.HasNextObject() DO
			IF ToXpMover(THIS^.fbMoversPresent.GetNextObject(),ipTempMover) AND_THEN ipTempMover.UtilityTcIoMover <> 0 THEN
				ipTempMover.UtilityTcIoMover.SetControllersOn(ControllersOn := stController);
			END_IF
		END_WHILE		
		nSeqEnabling := 25;		
		
		
		
	25: // Reset movers
		bWatchDogActive := TRUE;
		THIS^.fbMoversPresent.ResetIterator();
		WHILE THIS^.fbMoversPresent.HasNextObject() DO
			IF ToXpMover(THIS^.fbMoversPresent.GetNextObject(),ipTempMover) THEN
				hr := GetMostSignificant(hr, ipTempMover.Reset());
			END_IF
		END_WHILE
		
		IF CheckOk(hr) THEN 
			nSeqEnabling := 26;
		ELSE
			nSeqEnabling := 1000 + nSeqEnabling;
		END_IF		

	26: // Resetting movers
		bWatchDogActive := TRUE;
		THIS^.fbMoversPresent.ResetIterator();
		WHILE THIS^.fbMoversPresent.HasNextObject() DO
			IF ToXpMover(THIS^.fbMoversPresent.GetNextObject(),ipTempMover) THEN
				hr := GetMostSignificant(hr, ipTempMover.Feedback.HR);
			END_IF
		END_WHILE
		
		IF CheckOk(hr) THEN 
			nSeqEnabling := 30;
		ELSIF FAILED(hr) THEN
			nSeqEnabling := 1000 + nSeqEnabling;
		END_IF

		
		
	30: // Configure environment
		bWatchDogActive := TRUE;
		hr := ipEnvironment.Configure();
		
		IF CheckOk(hr) THEN 
			nSeqEnabling := 31;
		ELSE
			nSeqEnabling := 1000 + nSeqEnabling;
		END_IF	

	31: // Configuring environment
		bWatchDogActive := TRUE;
		hr := ipEnvironment.Feedback.HR;
		
		IF CheckOk(hr) THEN 
			nSeqEnabling := 50;
		ELSIF FAILED(hr) THEN
			nSeqEnabling := 1000 + nSeqEnabling;
		END_IF
		
		
	50: //Deside if or if not add enviroment to group
		bWatchDogActive := TRUE;
		IF XPlanarParameterlist.B_ADD_ENVIROMENT_TO_GROUP THEN
			nSeqEnabling := 51;
		ELSE
			nSeqEnabling := 70;
		END_IF
		
	51: // Add environment to group
		bWatchDogActive := TRUE;
		hr := ipEnvironment.AddToGroup(ipGroup);
		
		IF CheckOk(hr) THEN 
			nSeqEnabling := 52;
		ELSE
			nSeqEnabling := 1000 + nSeqEnabling;
		END_IF		

	52: // Adding environment to group
		bWatchDogActive := TRUE;
		hr := ipEnvironment.Feedback.HR;
		
		IF CheckOk(hr) THEN 
			nSeqEnabling := 70;
		ELSIF FAILED(hr) THEN
			nSeqEnabling := 1000 + nSeqEnabling;
		END_IF

		
	70: // Configure the tracks |
		bWatchDogActive := TRUE;
		THIS^.fbTracks.ResetIterator();
		WHILE THIS^.fbTracks.HasNextObject() DO
			IF ToXpTrack(THIS^.fbTracks.GetNextObject(),ipTempTrack) THEN
				hr := GetMostSignificant(hr, ipTempTrack.Configure());
			END_IF
		END_WHILE
		
		IF CheckOk(hr) THEN 
			nSeqEnabling := 71;
		ELSE
			nSeqEnabling := 1000 + nSeqEnabling;
		END_IF	
		
	71: // Configuring the tracks 
		bWatchDogActive := TRUE;
		THIS^.fbTracks.ResetIterator();
		WHILE THIS^.fbTracks.HasNextObject() DO
			IF ToXpTrack(THIS^.fbTracks.GetNextObject(),ipTempTrack) THEN
				hr := GetMostSignificant(hr, ipTempTrack.Configuring());
			END_IF
		END_WHILE
		
		IF CheckOk(hr) THEN 
			nSeqEnabling := 80;
		ELSIF FAILED(hr) THEN
			nSeqEnabling := 1000 + nSeqEnabling;
		END_IF	
		
		
	80: // Enable the tracks
		bWatchDogActive := TRUE;
		THIS^.fbTracks.ResetIterator();
		WHILE THIS^.fbTracks.HasNextObject() DO
			IF ToXpTrack(THIS^.fbTracks.GetNextObject(),ipTempTrack) THEN
				hr := GetMostSignificant(hr, ipTempTrack.Enable());
			END_IF
		END_WHILE
		
		IF CheckOk(hr) THEN 
			nSeqEnabling := 81;
		ELSE
			nSeqEnabling := 1000 + nSeqEnabling;
		END_IF		

	81: // Enabling the tracks
		bWatchDogActive := TRUE;
		THIS^.fbTracks.ResetIterator();
		WHILE THIS^.fbTracks.HasNextObject() DO
			IF ToXpTrack(THIS^.fbTracks.GetNextObject(),ipTempTrack) THEN
				hr := GetMostSignificant(hr, ipTempTrack.Feedback.HR);
			END_IF
		END_WHILE
		
		IF CheckOk(hr) THEN 
			nSeqEnabling := 90;
		ELSIF FAILED(hr) THEN
			nSeqEnabling := 1000 + nSeqEnabling;
		END_IF	
		
	90: //Deside if or if not add tracks to group
		bWatchDogActive := TRUE;
		IF XPlanarParameterlist.B_ADD_TRACKS_TO_GROUP THEN
			nSeqEnabling := 91;
		ELSE
			nSeqEnabling := 95;
		END_IF	
		
	91: // Add tracks to group
		bWatchDogActive := TRUE;
		THIS^.fbTracks.ResetIterator();
		WHILE THIS^.fbTracks.HasNextObject() DO
			IF ToXpTrack(THIS^.fbTracks.GetNextObject(),ipTempTrack) THEN
				hr := GetMostSignificant(hr, ipTempTrack.AddToGroup(ipGroup));
			END_IF
		END_WHILE
		
		IF CheckOk(hr) THEN 
			nSeqEnabling := 92;
		ELSE
			nSeqEnabling := 1000 + nSeqEnabling;
		END_IF	

	92: // Adding tracks to group
		bWatchDogActive := TRUE;
		THIS^.fbTracks.ResetIterator();
		WHILE THIS^.fbTracks.HasNextObject() DO
			IF ToXpTrack(THIS^.fbTracks.GetNextObject(),ipTempTrack) THEN
				hr := GetMostSignificant(hr, ipTempTrack.Feedback.HR);
			END_IF
		END_WHILE
		
		IF CheckOk(hr) THEN 
			nSeqEnabling := 95;
		ELSIF FAILED(hr) THEN
			nSeqEnabling := 1000 + nSeqEnabling;
		END_IF		
	
		
	95: // Enable movers
		//Enabling takes a relatively long time. To be a little quicker, the config is made before waiting for the enable.
		bWatchDogActive := TRUE;
		THIS^.fbMoversPresent.ResetIterator();
		WHILE THIS^.fbMoversPresent.HasNextObject() DO
			IF ToXpMover(THIS^.fbMoversPresent.GetNextObject(),ipTempMover) THEN
				hr := GetMostSignificant(hr, ipTempMover.Enable());
			END_IF
		END_WHILE
		
		IF CheckOk(hr) THEN 
			nSeqEnabling := 98;
		ELSE
			nSeqEnabling := 1000 + nSeqEnabling;
		END_IF			
		
		
	98: //Clear list of all paths
		bWatchDogActive := TRUE;
		THIS^.fbPaths.Clear();
		nSeqEnabling := 99;
		
	99: //Add all Stations to list of "Used" Stations, remove them later if not used
		THIS^.fbStationsUsed.Duplicate(THIS^.fbStationsAll);
		nSeqEnabling := 100;
		
	100..199: // Config Station
	(* All stations are always active to the same step to ensure that all data is available in the next step.
	   The following 100 steps are defined in the station. This makes overwriting easier *)
	   
		bWatchDogActive := TRUE;
		nSupSeq := nSeqEnabling - 100;
		THIS^.fbStationsUsed.ResetIterator();
		WHILE THIS^.fbStationsUsed.HasNextObject() DO
			IF ToXpStation(THIS^.fbStationsUsed.GetNextObject(),ipTempStation) THEN
				//Call this Methode whith seq 0->99, and wait each step until S_OK is returned. Call agaiin on S_Pending
				hr := GetMostSignificant(hr, ipTempStation.Configure(nSupSeq));
			END_IF
		END_WHILE	   
	   
	   
	   	IF CheckOk(hr) AND nSupSeq >= 99 THEN
			//All steps done 
			nSeqEnabling := 205;
		ELSIF FAILED(hr) THEN
			//Error
			nSeqEnabling := 1000 + nSeqEnabling;
		ELSIF CheckOk(hr) THEN 	 
			//active step is done, continous with next
			nSeqEnabling := nSeqEnabling + 1;
		END_IF	

	205: //Generate a list of all paths
		bWatchDogActive := TRUE;
		THIS^.fbStationsUsed.ResetIterator();
		WHILE THIS^.fbStationsUsed.HasNextObject() DO
			IF ToXpStation(THIS^.fbStationsUsed.GetNextObject(),ipTempStation) THEN
				THIS^.fbPaths.AddList(ipTempStation.PathsAhead);
			END_IF
		END_WHILE			
		
		nSeqEnabling := 211;
		
		
	211: // Enabling movers
		 //Enabling takes a relatively long time. To be a little quicker, the config is made before waiting for the enable.
		bWatchDogActive := TRUE;
		THIS^.fbMoversPresent.ResetIterator();
		WHILE THIS^.fbMoversPresent.HasNextObject() DO
			IF ToXpMover(THIS^.fbMoversPresent.GetNextObject(),ipTempMover) THEN
				hr := GetMostSignificant(hr, ipTempMover.Feedback.HR);
			END_IF
		END_WHILE
		
		IF CheckOk(hr) THEN 
			nSeqEnabling := 220;
		ELSIF FAILED(hr) THEN
			nSeqEnabling := 1000 + nSeqEnabling;
		END_IF	
		

	220: //Rotate A-Axis to zero
		bWatchDogActive := TRUE;
		THIS^.fbMoversPresent.ResetIterator();
		WHILE THIS^.fbMoversPresent.HasNextObject() DO
			IF ToXpMover(THIS^.fbMoversPresent.GetNextObject(),ipTempMover) THEN
				hr := GetMostSignificant(hr, ipTempMover.MoveA(0));
			END_IF
		END_WHILE
		
		IF CheckOk(hr) THEN 
			nSeqEnabling := 221;
		ELSE
			nSeqEnabling := 1000 + nSeqEnabling;
		END_IF	
		
	221: //Rotating A-Axis to Zero	
		bWatchDogActive := TRUE;		
		THIS^.fbMoversPresent.ResetIterator();
		WHILE THIS^.fbMoversPresent.HasNextObject() DO
			IF ToXpMover(THIS^.fbMoversPresent.GetNextObject(),ipTempMover) THEN
				hr := GetMostSignificant(hr, ipTempMover.Feedback.HR);
			END_IF
		END_WHILE
		
		IF CheckOk(hr) THEN 
			nSeqEnabling := 222;
		ELSIF FAILED(hr) THEN
			nSeqEnabling := 1000 + nSeqEnabling;
		END_IF	
		
		
		
	222: //Rotate B-Axis to zero
		bWatchDogActive := TRUE;
		THIS^.fbMoversPresent.ResetIterator();
		WHILE THIS^.fbMoversPresent.HasNextObject() DO
			IF ToXpMover(THIS^.fbMoversPresent.GetNextObject(),ipTempMover) THEN
				hr := GetMostSignificant(hr, ipTempMover.MoveB(0));
			END_IF
		END_WHILE
		
		IF CheckOk(hr) THEN 
			nSeqEnabling := 223;
		ELSE
			nSeqEnabling := 1000 + nSeqEnabling;
		END_IF	
		
	223: //Rotating B-Axis to zero
		bWatchDogActive := TRUE;			
		THIS^.fbMoversPresent.ResetIterator();
		WHILE THIS^.fbMoversPresent.HasNextObject() DO
			IF ToXpMover(THIS^.fbMoversPresent.GetNextObject(),ipTempMover) THEN
				hr := GetMostSignificant(hr, ipTempMover.Feedback.HR);
			END_IF
		END_WHILE
		
		IF CheckOk(hr) THEN 
			nSeqEnabling := 230;
		ELSIF FAILED(hr) THEN
			nSeqEnabling := 1000 + nSeqEnabling;
		END_IF		
		
				
		
	230: //Rotate C-Axis to "Zero" (to the next 90 degree pitch)
		bWatchDogActive := TRUE;
		THIS^.fbMoversPresent.ResetIterator();
		WHILE THIS^.fbMoversPresent.HasNextObject() DO
			IF ToXpMover(THIS^.fbMoversPresent.GetNextObject(),ipTempMover) THEN
				// Decide which 90 degree pitch is closer to the current position. If the remainder is greater than 45 degrees, then round up to the next 90 degree division.
				lrCRotationShortestPos := DINT_TO_LREAL(LREAL_TO_DINT(ipTempMover.PlanarMover.MCTOPLC.SET.SetPos.C / 90.0) * 90);
				lrCRotationShortestPos := MODABS(	lr_Value := lrCRotationShortestPos, 
													lr_Arg := ipTempMover.CAxisModulo);
				hr := GetMostSignificant(hr, ipTempMover.MoveC(	fPosition		:= lrCRotationShortestPos, 
																additionalTurns := 0,
																direction		:= Tc3_Mc3Definitions.MC_DIRECTION.mcDirectionShortestWay));
			END_IF
		END_WHILE
		
		IF CheckOk(hr) THEN 
			nSeqEnabling := 231;
		ELSE
			nSeqEnabling := 1000 + nSeqEnabling;
		END_IF	
		
		
	231: //Rotating C-Axis to Zero		
		bWatchDogActive := TRUE;	
		THIS^.fbMoversPresent.ResetIterator();
		WHILE THIS^.fbMoversPresent.HasNextObject() DO
			IF ToXpMover(THIS^.fbMoversPresent.GetNextObject(),ipTempMover) THEN
				hr := GetMostSignificant(hr, ipTempMover.Feedback.HR);
			END_IF
		END_WHILE
		
		IF CheckOk(hr) THEN 
			nSeqEnabling := 240;
		ELSIF FAILED(hr) THEN
			nSeqEnabling := 1000 + nSeqEnabling;
		END_IF	
		
			
	240: //Deside if or if not add movers to group
		bWatchDogActive := TRUE;
		IF XPlanarParameterlist.B_ADD_MOVERS_TO_GROUP THEN
			nSeqEnabling := 210;
		ELSE
			nSeqEnabling := 300;
		END_IF	
		
	241: // Add movers to group
		bWatchDogActive := TRUE;
		THIS^.fbMoversPresent.ResetIterator();
		WHILE THIS^.fbMoversPresent.HasNextObject() DO
			IF ToXpMover(THIS^.fbMoversPresent.GetNextObject(),ipTempMover) THEN
				hr := GetMostSignificant(hr, ipTempMover.AddToGroup(THIS^.ipGroup));
			END_IF
		END_WHILE
		
		IF CheckOk(hr) THEN 
			nSeqEnabling := 242;
		ELSE
			nSeqEnabling := 1000 + nSeqEnabling;
		END_IF	
		
		
